KUKA KRL program: EPS_2_25252_PD2_A_20250910061714.src

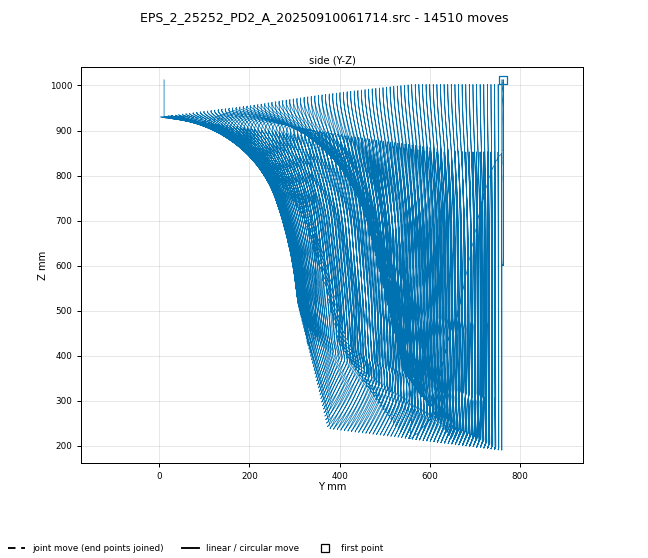
[picture p0: tool path of EPS_2_25252_PD2_A_20250910061714.src, 14510 of 14512 moves have a stored position in this frame; points joined in program order, loops and branches not executed]
&ACCESS RVP
&REL 4
&COMMENT QRS 19112012
&PARAM EDITMASK = *
DEF PART()
EXT BAS (BAS_COMMAND :IN,REAL :IN )
INT I
BAS (#INITMOV,0 )

;KUKA QRS Post kuka4.cps  Date:22-06-2017 !

File_ID=2827

QRS_PRE_INIT()

;Init var - Until changes are made in qrs_pre_init
Outlet_Square_prg=0
Inlet_1_Square_prg=0
Inlet_2_Square_prg=0
Inlet_3_Square_prg=0
Inlet_4_Square_prg=0
Inlet_5_Square_prg=0

Outlet_1={X 0.000, Y 562.000, Z 659.500, B 0.000, E1 0.000 }
Inlet_1={X 0.000, Y 675.710, Z 469.500, B 0.000, E1 90.000 }
Inlet_2={X 0.000, Y 612.000, Z 586.000, B 0.000, E1 180.000 }
Outlet_1_type=686
Inlet_1_type=366
Inlet_2_type=533
;QRS#1=Sidecore dimensions
;QRS#2=675-27" Concrete
;QRS#3=375-15" PVC SDR 35
;QRS#4=525-21" Concrete
;QRS#5=
;QRS#6=
;QRS#7=
;QRS#8=
;QRS#9=S306-38L
;QRS#10=20Y PSX
;QRS#11=S306-32
;QRS#12=
;QRS#13=
;QRS#14=
;QRS#15=
;QRS#16=1524x152x1448 4,75'
;QRS#17=EPS Height
;QRS#18=1002,5
;QRS#19=*
;QRS#20= UPDATED VERSION 22-06-2017
;QRS#21=*
Outlet_Square=0550
Inlet_1_Square=0250
Inlet_2_Square=0350
Inlet_3_Square=0
Inlet_4_Square=0
Inlet_5_Square=0
Mill_Square=1
Outlet_Square_Prg=265
Inlet_1_Square_prg=252
Inlet_2_Square_prg=263

QRS_INIT()

$ADVANCE=5

; T1
PTP {E1 177.625,E2 177.625}
PTP {X 0,Y 762.863,A -85,B 0,C 180,E1 177.625,E2 177.625,E3 0,E4 0,E5 0,E6 0}
QRS_SPEED_INIT()
LIN {X 0,Y 762.863,Z 1012.5,A -85,B 0,C 180,E1 177.625,E2 177.625,E3 0,E4 0,E5 0,E6 0} C_VEL
LIN {X 0,Y 762.863,Z 865.307,A -85,B 0,C 180,E1 177.625,E2 177.625} C_VEL
LIN {X 0,Y 762.863,Z 857.515,A -85,B 0,C 180,E1 177.625,E2 177.625} C_VEL
LIN {X 0,Y 762.89,Z 855.523,A -85,B 0,C 180,E1 177.789,E2 177.789} C_VEL
LIN {X 0,Y 763.311,Z 857.103,A -85,B 0,C 180,E1 179.062,E2 179.062} C_VEL
LIN {X 0,Y 763.552,Z 857.314,A -85,B 0,C 180,E1 179.437,E2 179.437} C_VEL
LIN {X 0,Y 763.78,Z 857.385,A -85,B 0,C 180,E1 180.187,E2 180.187} C_VEL
LIN {X 0,Y 763.382,Z 857.021,A -85,B 0,C 180,E1 180.938,E2 180.938} C_VEL
LIN {X 0,Y 763.064,Z 855.901,A -85,B 0,C 180,E1 181.878,E2 181.878} C_VEL
LIN {X 0,Y 763.224,Z 854.049,A -85,B 0,C 180,E1 182.816,E2 182.816} C_VEL
LIN {X 0,Y 763.674,Z 851.777,A -85,B 0,C 180,E1 183.621,E2 183.621} C_VEL
LIN {X 0,Y 763.795,Z 849.977,A -85,B 0,C 180,E1 184.156,E2 184.156} C_VEL
LIN {X 0,Y 763.342,Z 846.94,A -85,B 0,C 180,E1 184.931,E2 184.931} C_VEL
LIN {X 0,Y 763.012,Z 843.639,A -85,B 0,C 180,E1 185.64,E2 185.64} C_VEL
LIN {X 0,Y 763,Z 839.822,A -85,B 0,C 180,E1 186.347,E2 186.347} C_VEL
LIN {X 0,Y 763.321,Z 835.459,A -85,B 0,C 180,E1 187.053,E2 187.053} C_VEL
LIN {X 0,Y 763.757,Z 830.521,A -85,B 0,C 180,E1 187.758,E2 187.758} C_VEL
LIN {X 0,Y 763.804,Z 826.923,A -85,B 0,C 180,E1 188.231,E2 188.231} C_VEL
LIN {X 0,Y 763.447,Z 819.835,A -85,B 0,C 180,E1 189.065,E2 189.065} C_VEL
LIN {X 0,Y 763.299,Z 814.185,A -85,B 0,C 180,E1 189.661,E2 189.661} C_VEL
LIN {X 0,Y 763.415,Z 807.963,A -85,B 0,C 180,E1 190.255,E2 190.255} C_VEL
LIN {X 0,Y 763.624,Z 802.554,A -85,B 0,C 180,E1 190.729,E2 190.729} C_VEL
LIN {X 0,Y 763.851,Z 795.117,A -85,B 0,C 180,E1 191.322,E2 191.322} C_VEL
LIN {X 0,Y 763.76,Z 788.602,A -85,B 0,C 180,E1 191.802,E2 191.802} C_VEL
LIN {X 0,Y 763.573,Z 781.49,A -85,B 0,C 180,E1 192.284,E2 192.284} C_VEL
LIN {X 0,Y 763.481,Z 774.931,A -85,B 0,C 180,E1 192.694,E2 192.694} C_VEL
LIN {X 0,Y 763.571,Z 767.346,A -85,B 0,C 180,E1 193.125,E2 193.125} C_VEL
LIN {X 0,Y 763.752,Z 758.954,A -85,B 0,C 180,E1 193.555,E2 193.555} C_VEL
LIN {X 0,Y 763.785,Z 751.25,A -85,B 0,C 180,E1 193.917,E2 193.917} C_VEL
LIN {X 0,Y 763.828,Z 741.459,A -85,B 0,C 180,E1 194.328,E2 194.328} C_VEL
LIN {X 0,Y 763.759,Z 733.415,A -85,B 0,C 180,E1 194.632,E2 194.632} C_VEL
LIN {X 0,Y 763.747,Z 724.359,A -85,B 0,C 180,E1 194.936,E2 194.936} C_VEL
LIN {X 0,Y 763.826,Z 715.053,A -85,B 0,C 180,E1 195.207,E2 195.207} C_VEL
LIN {X 0,Y 763.801,Z 705.091,A -85,B 0,C 180,E1 195.458,E2 195.458} C_VEL
LIN {X 0,Y 763.852,Z 696.194,A -85,B 0,C 180,E1 195.647,E2 195.647} C_VEL
LIN {X 0,Y 763.86,Z 686.714,A -85,B 0,C 180,E1 195.814,E2 195.814} C_VEL
LIN {X 0,Y 763.829,Z 678.167,A -85,B 0,C 180,E1 195.936,E2 195.936} C_VEL
LIN {X 0,Y 763.809,Z 660.489,A -85,B 0,C 180,E1 196.119,E2 196.119} C_VEL
LIN {X 0,Y 763.591,Z 638.669,A -85,B 0,C 180,E1 196.333,E2 196.333} C_VEL
LIN {X 0,Y 763.668,Z 601.31,A -85,B 0,C 180,E1 197.602,E2 197.602} C_VEL
LIN {X 0,Y 763.856,Z 601.31,A -85,B 0,C 180,E1 200.095,E2 200.095} C_VEL
LIN {X 0,Y 763.798,Z 601.31,A -85,B 0,C 180,E1 208.326,E2 208.326} C_VEL
LIN {X 0,Y 762.387,Z 601.31,A -85,B 0,C 180,E1 210.541,E2 210.541} C_VEL
LIN {X 0,Y 762.703,Z 601.31,A -85,B 0,C 180,E1 214.993,E2 214.993} C_VEL
LIN {X 0,Y 763.707,Z 601.31,A -85,B 0,C 180,E1 216.696,E2 216.696} C_VEL
LIN {X 0,Y 763.72,Z 601.31,A -85,B 0,C 180,E1 224.719,E2 224.719} C_VEL
LIN {X 0,Y 763.504,Z 601.31,A -85,B 0,C 180,E1 225.265,E2 225.265} C_VEL
LIN {X 0,Y 762.431,Z 601.31,A -85,B 0,C 180,E1 230.388,E2 230.388} C_VEL
LIN {X 0,Y 763.803,Z 601.31,A -85,B 0,C 180,E1 232.744,E2 232.744} C_VEL
LIN {X 0,Y 763.78,Z 601.31,A -85,B 0,C 180,E1 239.845,E2 239.845} C_VEL
LIN {X 0,Y 763.759,Z 601.31,A -85,B 0,C 180,E1 240.061,E2 240.061} C_VEL
LIN {X 0,Y 763.232,Z 601.31,A -85,B 0,C 180,E1 240.149,E2 240.149} C_VEL
LIN {X 0,Y 763.551,Z 649.404,A -85,B 0,C 180,E1 240.674,E2 240.674} C_VEL
LIN {X 0,Y 763.815,Z 684.428,A -85,B 0,C 180,E1 241.063,E2 241.063} C_VEL
LIN {X 0,Y 763.833,Z 699.23,A -85,B 0,C 180,E1 241.258,E2 241.258} C_VEL
LIN {X 0,Y 763.72,Z 715.993,A -85,B 0,C 180,E1 241.54,E2 241.54} C_VEL
LIN {X 0,Y 763.487,Z 727.212,A -85,B 0,C 180,E1 241.761,E2 241.761} C_VEL
LIN {X 0,Y 763.725,Z 739.829,A -85,B 0,C 180,E1 242.069,E2 242.069} C_VEL
LIN {X 0,Y 763.771,Z 748.863,A -85,B 0,C 180,E1 242.303,E2 242.303} C_VEL
LIN {X 0,Y 763.77,Z 763.638,A -85,B 0,C 180,E1 242.732,E2 242.732} C_VEL
LIN {X 0,Y 763.697,Z 781.216,A -85,B 0,C 180,E1 243.321,E2 243.321} C_VEL
LIN {X 0,Y 763.6,Z 789.955,A -85,B 0,C 180,E1 243.645,E2 243.645} C_VEL
LIN {X 0,Y 763.691,Z 798.571,A -85,B 0,C 180,E1 243.99,E2 243.99} C_VEL
LIN {X 0,Y 763.619,Z 811.78,A -85,B 0,C 180,E1 244.551,E2 244.551} C_VEL
LIN {X 0,Y 763.589,Z 826.422,A -85,B 0,C 180,E1 245.241,E2 245.241} C_VEL
LIN {X 0,Y 763.713,Z 840.578,A -85,B 0,C 180,E1 245.981,E2 245.981} C_VEL
LIN {X 0,Y 763.688,Z 854.073,A -85,B 0,C 180,E1 246.747,E2 246.747} C_VEL
LIN {X 0,Y 763.544,Z 866.427,A -85,B 0,C 180,E1 247.506,E2 247.506} C_VEL
LIN {X 0,Y 763.324,Z 879.551,A -85,B 0,C 180,E1 248.385,E2 248.385} C_VEL
LIN {X 0,Y 763.405,Z 891.553,A -85,B 0,C 180,E1 249.267,E2 249.267} C_VEL
LIN {X 0,Y 763.694,Z 903.235,A -85,B 0,C 180,E1 250.204,E2 250.204} C_VEL
LIN {X 0,Y 763.727,Z 910.839,A -85,B 0,C 180,E1 250.857,E2 250.857} C_VEL
LIN {X 0,Y 763.444,Z 918.944,A -85,B 0,C 180,E1 251.586,E2 251.586} C_VEL
LIN {X 0,Y 763.19,Z 925.901,A -85,B 0,C 180,E1 252.243,E2 252.243} C_VEL
LIN {X 0,Y 763.133,Z 935.473,A -85,B 0,C 180,E1 253.224,E2 253.224} C_VEL
LIN {X 0,Y 763.43,Z 944.365,A -85,B 0,C 180,E1 254.22,E2 254.22} C_VEL
LIN {X 0,Y 763.797,Z 951.479,A -85,B 0,C 180,E1 255.09,E2 255.09} C_VEL
LIN {X 0,Y 763.66,Z 955.119,A -85,B 0,C 180,E1 255.556,E2 255.556} C_VEL
LIN {X 0,Y 763.118,Z 962.759,A -85,B 0,C 180,E1 256.586,E2 256.586} C_VEL
LIN {X 0,Y 762.806,Z 970.221,A -85,B 0,C 180,E1 257.703,E2 257.703} C_VEL
LIN {X 0,Y 763.093,Z 977.341,A -85,B 0,C 180,E1 258.905,E2 258.905} C_VEL
LIN {X 0,Y 763.744,Z 983.625,A -85,B 0,C 180,E1 260.107,E2 260.107} C_VEL
LIN {X 0,Y 763.847,Z 984.734,A -85,B 0,C 180,E1 260.346,E2 260.346} C_VEL
LIN {X 0,Y 763.274,Z 989.117,A -85,B 0,C 180,E1 261.289,E2 261.289} C_VEL
LIN {X 0,Y 762.776,Z 993.85,A -85,B 0,C 180,E1 262.468,E2 262.468} C_VEL
LIN {X 0,Y 762.955,Z 998.504,A -85,B 0,C 180,E1 263.888,E2 263.888} C_VEL
LIN {X 0,Y 763.445,Z 1001.065,A -85,B 0,C 180,E1 264.834,E2 264.834} C_VEL
LIN {X 0,Y 763.752,Z 1002.127,A -85,B 0,C 180,E1 265.307,E2 265.307} C_VEL
LIN {X 0,Y 763.413,Z 1004.112,A -85,B 0,C 180,E1 266.245,E2 266.245} C_VEL
LIN {X 0,Y 762.878,Z 1005.536,A -85,B 0,C 180,E1 267.183,E2 267.183} C_VEL
LIN {X 0,Y 762.652,Z 1006.74,A -85,B 0,C 180,E1 268.315,E2 268.315} C_VEL
LIN {X 0,Y 762.792,Z 1007.219,A -85,B 0,C 180,E1 269.061,E2 269.061} C_VEL
LIN {X 0,Y 763.864,Z 1007.171,A -85,B 0,C 180,E1 270.937,E2 270.937} C_VEL
LIN {X 0,Y 763.506,Z 1006.761,A -85,B 0,C 180,E1 271.626,E2 271.626} C_VEL
LIN {X 0,Y 763.098,Z 1005.877,A -85,B 0,C 180,E1 272.585,E2 272.585} C_VEL
LIN {X 0,Y 763.034,Z 1004.125,A -85,B 0,C 180,E1 273.756,E2 273.756} C_VEL
LIN {X 0,Y 763.619,Z 1001.06,A -85,B 0,C 180,E1 275.164,E2 275.164} C_VEL
LIN {X 0,Y 763.871,Z 999.763,A -85,B 0,C 180,E1 275.633,E2 275.633} C_VEL
LIN {X 0,Y 763.32,Z 997.027,A -85,B 0,C 180,E1 276.581,E2 276.581} C_VEL
LIN {X 0,Y 762.845,Z 993.851,A -85,B 0,C 180,E1 277.531,E2 277.531} C_VEL
LIN {X 0,Y 762.834,Z 988.065,A -85,B 0,C 180,E1 278.953,E2 278.953} C_VEL
LIN {X 0,Y 763.409,Z 982.441,A -85,B 0,C 180,E1 280.135,E2 280.135} C_VEL
LIN {X 0,Y 763.842,Z 978.617,A -85,B 0,C 180,E1 280.845,E2 280.845} C_VEL
LIN {X 0,Y 763.475,Z 974.56,A -85,B 0,C 180,E1 281.567,E2 281.567} C_VEL
LIN {X 0,Y 762.978,Z 968.584,A -85,B 0,C 180,E1 282.553,E2 282.553} C_VEL
LIN {X 0,Y 762.85,Z 960.441,A -85,B 0,C 180,E1 283.748,E2 283.748} C_VEL
LIN {X 0,Y 763.269,Z 952.013,A -85,B 0,C 180,E1 284.856,E2 284.856} C_VEL
LIN {X 0,Y 763.798,Z 943.48,A -85,B 0,C 180,E1 285.876,E2 285.876} C_VEL
LIN {X 0,Y 763.424,Z 933.185,A -85,B 0,C 180,E1 287.014,E2 287.014} C_VEL
LIN {X 0,Y 763.153,Z 923.436,A -85,B 0,C 180,E1 288.004,E2 288.004} C_VEL
LIN {X 0,Y 763.309,Z 911.702,A -85,B 0,C 180,E1 289.081,E2 289.081} C_VEL
LIN {X 0,Y 763.648,Z 901.038,A -85,B 0,C 180,E1 289.977,E2 289.977} C_VEL
LIN {X 0,Y 763.74,Z 891.15,A -85,B 0,C 180,E1 290.756,E2 290.756} C_VEL
LIN {X 0,Y 763.498,Z 877.794,A -85,B 0,C 180,E1 291.733,E2 291.733} C_VEL
LIN {X 0,Y 763.446,Z 864.411,A -85,B 0,C 180,E1 292.624,E2 292.624} C_VEL
LIN {X 0,Y 763.624,Z 850.805,A -85,B 0,C 180,E1 293.446,E2 293.446} C_VEL
LIN {X 0,Y 763.68,Z 836.999,A -85,B 0,C 180,E1 294.213,E2 294.213} C_VEL
LIN {X 0,Y 763.702,Z 822.332,A -85,B 0,C 180,E1 294.955,E2 294.955} C_VEL
LIN {X 0,Y 763.621,Z 807.81,A -85,B 0,C 180,E1 295.625,E2 295.625} C_VEL
LIN {X 0,Y 763.676,Z 793.458,A -85,B 0,C 180,E1 296.221,E2 296.221} C_VEL
LIN {X 0,Y 763.623,Z 777.576,A -85,B 0,C 180,E1 296.812,E2 296.812} C_VEL
LIN {X 0,Y 763.541,Z 771.61,A -85,B 0,C 180,E1 297.013,E2 297.013} C_VEL
LIN {X 0,Y 763.734,Z 760.339,A -85,B 0,C 180,E1 297.368,E2 297.368} C_VEL
LIN {X 0,Y 763.776,Z 744.554,A -85,B 0,C 180,E1 297.812,E2 297.812} C_VEL
LIN {X 0,Y 763.736,Z 728.036,A -85,B 0,C 180,E1 298.212,E2 298.212} C_VEL
LIN {X 0,Y 763.451,Z 711.795,A -85,B 0,C 180,E1 298.55,E2 298.55} C_VEL
LIN {X 0,Y 763.682,Z 694.79,A -85,B 0,C 180,E1 298.813,E2 298.813} C_VEL
LIN {X 0,Y 763.667,Z 674.795,A -85,B 0,C 180,E1 299.053,E2 299.053} C_VEL
LIN {X 0,Y 763.245,Z 602.276,A -85,B 0,C 180,E1 299.838,E2 299.838} C_VEL
LIN {X 0,Y 763.307,Z 601.31,A -85,B 0,C 180,E1 299.858,E2 299.858} C_VEL
LIN {X 0,Y 763.723,Z 601.31,A -85,B 0,C 180,E1 299.929,E2 299.929} C_VEL
LIN {X 0,Y 763.822,Z 601.31,A -85,B 0,C 180,E1 300.149,E2 300.149} C_VEL
LIN {X 0,Y 763.79,Z 601.31,A -85,B 0,C 180,E1 304.936,E2 304.936} C_VEL
LIN {X 0,Y 762.495,Z 601.31,A -85,B 0,C 180,E1 309.732,E2 309.732} C_VEL
LIN {X 0,Y 763.786,Z 601.31,A -85,B 0,C 180,E1 312.132,E2 312.132} C_VEL
LIN {X 0,Y 763.614,Z 601.31,A -85,B 0,C 180,E1 312.57,E2 312.57} C_VEL
LIN {X 0,Y 763.854,Z 601.31,A -85,B 0,C 180,E1 320.259,E2 320.259} C_VEL
LIN {X 0,Y 763.733,Z 601.31,A -85,B 0,C 180,E1 326.566,E2 326.566} C_VEL
LIN {X 0,Y 763.485,Z 601.31,A -85,B 0,C 180,E1 327.305,E2 327.305} C_VEL
LIN {X 0,Y 763.791,Z 601.31,A -85,B 0,C 180,E1 333.783,E2 333.783} C_VEL
LIN {X 0,Y 763.817,Z 601.31,A -85,B 0,C 180,E1 341.889,E2 341.889} C_VEL
LIN {X 0,Y 763.825,Z 601.31,A -85,B 0,C 180,E1 349.632,E2 349.632} C_VEL
LIN {X 0,Y 763.858,Z 601.31,A -85,B 0,C 180,E1 357.187,E2 357.187} C_VEL
LIN {X 0,Y 763.862,Z 601.31,A -85,B 0,C 180,E1 364.692,E2 364.692} C_VEL
LIN {X 0,Y 763.839,Z 601.31,A -85,B 0,C 180,E1 372.28,E2 372.28} C_VEL
LIN {X 0,Y 763.83,Z 601.31,A -85,B 0,C 180,E1 380.095,E2 380.095} C_VEL
LIN {X 0,Y 763.817,Z 601.31,A -85,B 0,C 180,E1 388.325,E2 388.325} C_VEL
LIN {X 0,Y 762.039,Z 601.31,A -85,B 0,C 180,E1 393.241,E2 393.241} C_VEL
LIN {X 0,Y 762.697,Z 601.31,A -85,B 0,C 180,E1 394.994,E2 394.994} C_VEL
LIN {X 0,Y 763.698,Z 601.31,A -85,B 0,C 180,E1 396.695,E2 396.695} C_VEL
LIN {X 0,Y 763.727,Z 601.31,A -85,B 0,C 180,E1 404.718,E2 404.718} C_VEL
LIN {X 0,Y 763.509,Z 601.31,A -85,B 0,C 180,E1 405.266,E2 405.266} C_VEL
LIN {X 0,Y 762.413,Z 601.31,A -85,B 0,C 180,E1 410.39,E2 410.39} C_VEL
LIN {X 0,Y 763.781,Z 601.31,A -85,B 0,C 180,E1 412.743,E2 412.743} C_VEL
LIN {X 0,Y 763.812,Z 601.31,A -85,B 0,C 180,E1 419.522,E2 419.522} C_VEL
LIN {X 0,Y 763.566,Z 601.31,A -85,B 0,C 180,E1 426.715,E2 426.715} C_VEL
LIN {X 0,Y 763.593,Z 601.31,A -85,B 0,C 180,E1 427.187,E2 427.187} C_VEL
LIN {X 0,Y 762.639,Z 601.31,A -85,B 0,C 180,E1 427.3,E2 427.3} C_VEL
LIN {X 0,Y 763.453,Z 613.717,A -85,B 0,C 180,E1 427.49,E2 427.49} C_VEL
LIN {X 0,Y 763.724,Z 626.926,A -85,B 0,C 180,E1 427.717,E2 427.717} C_VEL
LIN {X 0,Y 763.789,Z 639.679,A -85,B 0,C 180,E1 427.979,E2 427.979} C_VEL
LIN {X 0,Y 763.776,Z 651.564,A -85,B 0,C 180,E1 428.263,E2 428.263} C_VEL
LIN {X 0,Y 763.642,Z 664.747,A -85,B 0,C 180,E1 428.628,E2 428.628} C_VEL
LIN {X 0,Y 763.763,Z 676.879,A -85,B 0,C 180,E1 429.02,E2 429.02} C_VEL
LIN {X 0,Y 763.692,Z 689.935,A -85,B 0,C 180,E1 429.494,E2 429.494} C_VEL
LIN {X 0,Y 763.704,Z 701.321,A -85,B 0,C 180,E1 429.958,E2 429.958} C_VEL
LIN {X 0,Y 763.78,Z 713.403,A -85,B 0,C 180,E1 430.507,E2 430.507} C_VEL
LIN {X 0,Y 763.744,Z 724.924,A -85,B 0,C 180,E1 431.083,E2 431.083} C_VEL
LIN {X 0,Y 763.624,Z 736.787,A -85,B 0,C 180,E1 431.738,E2 431.738} C_VEL
LIN {X 0,Y 763.515,Z 745.388,A -85,B 0,C 180,E1 432.251,E2 432.251} C_VEL
LIN {X 0,Y 763.577,Z 756.581,A -85,B 0,C 180,E1 432.989,E2 432.989} C_VEL
LIN {X 0,Y 763.781,Z 766.757,A -85,B 0,C 180,E1 433.728,E2 433.728} C_VEL
LIN {X 0,Y 763.734,Z 775.073,A -85,B 0,C 180,E1 434.376,E2 434.376} C_VEL
LIN {X 0,Y 763.38,Z 783.89,A -85,B 0,C 180,E1 435.117,E2 435.117} C_VEL
LIN {X 0,Y 763.135,Z 792.692,A -85,B 0,C 180,E1 435.929,E2 435.929} C_VEL
LIN {X 0,Y 763.213,Z 800.042,A -85,B 0,C 180,E1 436.669,E2 436.669} C_VEL
LIN {X 0,Y 763.601,Z 808.027,A -85,B 0,C 180,E1 437.558,E2 437.558} C_VEL
LIN {X 0,Y 763.841,Z 813.343,A -85,B 0,C 180,E1 438.199,E2 438.199} C_VEL
LIN {X 0,Y 763.358,Z 820.655,A -85,B 0,C 180,E1 439.148,E2 439.148} C_VEL
LIN {X 0,Y 762.982,Z 827.171,A -85,B 0,C 180,E1 440.097,E2 440.097} C_VEL
LIN {X 0,Y 763.039,Z 832.95,A -85,B 0,C 180,E1 441.049,E2 441.049} C_VEL
LIN {X 0,Y 763.49,Z 838.043,A -85,B 0,C 180,E1 442.003,E2 442.003} C_VEL
LIN {X 0,Y 763.847,Z 841.371,A -85,B 0,C 180,E1 442.716,E2 442.716} C_VEL
LIN {X 0,Y 763.45,Z 844.408,A -85,B 0,C 180,E1 443.42,E2 443.42} C_VEL
LIN {X 0,Y 763.18,Z 846.302,A -85,B 0,C 180,E1 443.89,E2 443.89} C_VEL
LIN {X 0,Y 762.856,Z 849.53,A -85,B 0,C 180,E1 444.831,E2 444.831} C_VEL
LIN {X 0,Y 763.052,Z 852.685,A -85,B 0,C 180,E1 445.96,E2 445.96} C_VEL
LIN {X 0,Y 763.753,Z 855.112,A -85,B 0,C 180,E1 447.186,E2 447.186} C_VEL
LIN {X 0,Y 763.548,Z 856.237,A -85,B 0,C 180,E1 447.937,E2 447.937} C_VEL
LIN {X 0,Y 762.891,Z 857.232,A -85,B 0,C 180,E1 449.062,E2 449.062} C_VEL
LIN {X 0,Y 762.996,Z 857.194,A -85,B 0,C 180,E1 450.939,E2 450.939} C_VEL
LIN {X 0,Y 763.457,Z 856.519,A -85,B 0,C 180,E1 451.689,E2 451.689} C_VEL
LIN {X 0,Y 763.608,Z 854.985,A -85,B 0,C 180,E1 452.814,E2 452.814} C_VEL
LIN {X 0,Y 762.972,Z 852.552,A -85,B 0,C 180,E1 454.001,E2 454.001} C_VEL
LIN {X 0,Y 762.867,Z 850.661,A -85,B 0,C 180,E1 454.698,E2 454.698} C_VEL
LIN {X 0,Y 763.096,Z 847.645,A -85,B 0,C 180,E1 455.639,E2 455.639} C_VEL
LIN {X 0,Y 763.607,Z 844.044,A -85,B 0,C 180,E1 456.578,E2 456.578} C_VEL
LIN {X 0,Y 763.863,Z 842.053,A -85,B 0,C 180,E1 457.048,E2 457.048} C_VEL
LIN {X 0,Y 763.388,Z 837.561,A -85,B 0,C 180,E1 457.999,E2 457.999} C_VEL
LIN {X 0,Y 763.01,Z 832.407,A -85,B 0,C 180,E1 458.952,E2 458.952} C_VEL
LIN {X 0,Y 763.055,Z 826.56,A -85,B 0,C 180,E1 459.902,E2 459.902} C_VEL
LIN {X 0,Y 763.496,Z 819.973,A -85,B 0,C 180,E1 460.85,E2 460.85} C_VEL
LIN {X 0,Y 763.851,Z 814.56,A -85,B 0,C 180,E1 461.561,E2 461.561} C_VEL
LIN {X 0,Y 763.411,Z 805.949,A -85,B 0,C 180,E1 462.592,E2 462.592} C_VEL
LIN {X 0,Y 763.116,Z 797.827,A -85,B 0,C 180,E1 463.469,E2 463.469} C_VEL
LIN {X 0,Y 763.167,Z 790.215,A -85,B 0,C 180,E1 464.219,E2 464.219} C_VEL
LIN {X 0,Y 763.551,Z 780.772,A -85,B 0,C 180,E1 465.06,E2 465.06} C_VEL
LIN {X 0,Y 763.786,Z 772.241,A -85,B 0,C 180,E1 465.759,E2 465.759} C_VEL
LIN {X 0,Y 763.672,Z 763.931,A -85,B 0,C 180,E1 466.397,E2 466.397} C_VEL
LIN {X 0,Y 763.452,Z 753.435,A -85,B 0,C 180,E1 467.136,E2 467.136} C_VEL
LIN {X 0,Y 763.432,Z 742.882,A -85,B 0,C 180,E1 467.813,E2 467.813} C_VEL
LIN {X 0,Y 763.629,Z 732.669,A -85,B 0,C 180,E1 468.408,E2 468.408} C_VEL
LIN {X 0,Y 763.748,Z 721.763,A -85,B 0,C 180,E1 468.99,E2 468.99} C_VEL
LIN {X 0,Y 763.776,Z 710.571,A -85,B 0,C 180,E1 469.537,E2 469.537} C_VEL
LIN {X 0,Y 763.679,Z 697.818,A -85,B 0,C 180,E1 470.1,E2 470.1} C_VEL
LIN {X 0,Y 763.694,Z 685.483,A -85,B 0,C 180,E1 470.584,E2 470.584} C_VEL
LIN {X 0,Y 763.756,Z 672.801,A -85,B 0,C 180,E1 471.024,E2 471.024} C_VEL
LIN {X 0,Y 763.656,Z 660.443,A -85,B 0,C 180,E1 471.407,E2 471.407} C_VEL
LIN {X 0,Y 763.818,Z 647.246,A -85,B 0,C 180,E1 471.753,E2 471.753} C_VEL
LIN {X 0,Y 763.833,Z 634.146,A -85,B 0,C 180,E1 472.049,E2 472.049} C_VEL
LIN {X 0,Y 763.831,Z 621.273,A -85,B 0,C 180,E1 472.29,E2 472.29} C_VEL
LIN {X 0,Y 763.727,Z 607.963,A -85,B 0,C 180,E1 472.492,E2 472.492} C_VEL
LIN {X 0,Y 763.443,Z 601.78,A -85,B 0,C 180,E1 472.574,E2 472.574} C_VEL
LIN {X 0,Y 763.321,Z 601.31,A -85,B 0,C 180,E1 472.594,E2 472.594} C_VEL
LIN {X 0,Y 763.424,Z 601.31,A -85,B 0,C 180,E1 472.759,E2 472.759} C_VEL
LIN {X 0,Y 762.937,Z 601.31,A -85,B 0,C 180,E1 476.249,E2 476.249} C_VEL
LIN {X 0,Y 763.845,Z 601.31,A -85,B 0,C 180,E1 478.324,E2 478.324} C_VEL
LIN {X 0,Y 762.047,Z 601.31,A -85,B 0,C 180,E1 483.242,E2 483.242} C_VEL
LIN {X 0,Y 762.711,Z 601.31,A -85,B 0,C 180,E1 484.993,E2 484.993} C_VEL
LIN {X 0,Y 763.72,Z 601.31,A -85,B 0,C 180,E1 486.697,E2 486.697} C_VEL
LIN {X 0,Y 763.748,Z 601.31,A -85,B 0,C 180,E1 494.717,E2 494.717} C_VEL
LIN {X 0,Y 763.532,Z 601.31,A -85,B 0,C 180,E1 495.267,E2 495.267} C_VEL
LIN {X 0,Y 762.433,Z 601.31,A -85,B 0,C 180,E1 500.388,E2 500.388} C_VEL
LIN {X 0,Y 763.807,Z 601.31,A -85,B 0,C 180,E1 502.744,E2 502.744} C_VEL
LIN {X 0,Y 763.794,Z 601.31,A -85,B 0,C 180,E1 509.521,E2 509.521} C_VEL
LIN {X 0,Y 763.794,Z 601.31,A -85,B 0,C 180,E1 515.855,E2 515.855} C_VEL
LIN {X 0,Y 763.311,Z 601.31,A -85,B 0,C 180,E1 522.34,E2 522.34} C_VEL
LIN {X 0,Y 763.596,Z 630.997,A -85,B 0,C 180,E1 523.503,E2 523.503} C_VEL
LIN {X 0,Y 763.782,Z 675.397,A -85,B 0,C 180,E1 523.941,E2 523.941} C_VEL
LIN {X 0,Y 763.733,Z 684.643,A -85,B 0,C 180,E1 524.063,E2 524.063} C_VEL
LIN {X 0,Y 763.831,Z 693.752,A -85,B 0,C 180,E1 524.217,E2 524.217} C_VEL
LIN {X 0,Y 763.791,Z 702.752,A -85,B 0,C 180,E1 524.399,E2 524.399} C_VEL
LIN {X 0,Y 763.731,Z 711.65,A -85,B 0,C 180,E1 524.611,E2 524.611} C_VEL
LIN {X 0,Y 763.755,Z 719.441,A -85,B 0,C 180,E1 524.825,E2 524.825} C_VEL
LIN {X 0,Y 763.831,Z 729.06,A -85,B 0,C 180,E1 525.129,E2 525.129} C_VEL
LIN {X 0,Y 763.796,Z 737.568,A -85,B 0,C 180,E1 525.43,E2 525.43} C_VEL
LIN {X 0,Y 763.775,Z 746.635,A -85,B 0,C 180,E1 525.793,E2 525.793} C_VEL
LIN {X 0,Y 763.751,Z 755.527,A -85,B 0,C 180,E1 526.19,E2 526.19} C_VEL
LIN {X 0,Y 763.567,Z 763.547,A -85,B 0,C 180,E1 526.584,E2 526.584} C_VEL
LIN {X 0,Y 763.449,Z 770.453,A -85,B 0,C 180,E1 526.955,E2 526.955} C_VEL
LIN {X 0,Y 763.526,Z 778.468,A -85,B 0,C 180,E1 527.432,E2 527.432} C_VEL
LIN {X 0,Y 763.752,Z 786.449,A -85,B 0,C 180,E1 527.958,E2 527.958} C_VEL
LIN {X 0,Y 763.854,Z 793.148,A -85,B 0,C 180,E1 528.439,E2 528.439} C_VEL
LIN {X 0,Y 763.691,Z 799.305,A -85,B 0,C 180,E1 528.914,E2 528.914} C_VEL
LIN {X 0,Y 763.419,Z 806.315,A -85,B 0,C 180,E1 529.507,E2 529.507} C_VEL
LIN {X 0,Y 763.312,Z 811.472,A -85,B 0,C 180,E1 529.982,E2 529.982} C_VEL
LIN {X 0,Y 763.402,Z 817.368,A -85,B 0,C 180,E1 530.578,E2 530.578} C_VEL
LIN {X 0,Y 763.605,Z 821.734,A -85,B 0,C 180,E1 531.056,E2 531.056} C_VEL
LIN {X 0,Y 763.881,Z 827.607,A -85,B 0,C 180,E1 531.77,E2 531.77} C_VEL
LIN {X 0,Y 763.496,Z 832.846,A -85,B 0,C 180,E1 532.476,E2 532.476} C_VEL
LIN {X 0,Y 763.198,Z 836.057,A -85,B 0,C 180,E1 532.946,E2 532.946} C_VEL
LIN {X 0,Y 762.985,Z 840.331,A -85,B 0,C 180,E1 533.652,E2 533.652} C_VEL
LIN {X 0,Y 763.11,Z 844.072,A -85,B 0,C 180,E1 534.361,E2 534.361} C_VEL
LIN {X 0,Y 763.363,Z 846.268,A -85,B 0,C 180,E1 534.834,E2 534.834} C_VEL
LIN {X 0,Y 763.807,Z 849.501,A -85,B 0,C 180,E1 535.624,E2 535.624} C_VEL
LIN {X 0,Y 763.791,Z 850.603,A -85,B 0,C 180,E1 535.941,E2 535.941} C_VEL
LIN {X 0,Y 763.396,Z 852.627,A -85,B 0,C 180,E1 536.571,E2 536.571} C_VEL
LIN {X 0,Y 763.05,Z 854.257,A -85,B 0,C 180,E1 537.184,E2 537.184} C_VEL
LIN {X 0,Y 762.89,Z 855.523,A -85,B 0,C 180,E1 537.789,E2 537.789} C_VEL
LIN {X 0,Y 762.867,Z 857.499,A -85,B 0,C 180,E1 537.916,E2 537.916} C_VEL
LIN {X 0,Y 762.867,Z 1012.5,A -85,B 0,C 180,E1 537.916,E2 537.916} C_VEL
LIN {X 0,Y 762.867,Z 1012.5,A -85,B 0,C 180,E1 537.916,E2 537.916}

QRS_NEXT_CUT()
PTP {E1 537.186,E2 537.186}
PTP {X 0,Y 759.911,A -85,B 0,C 180,E1 537.186,E2 537.186,E3 0,E4 0,E5 0,E6 0}
QRS_SPEED_INIT()
LIN {X 0,Y 759.911,Z 1012.5,A -85,B 0,C 180,E1 537.186,E2 537.186,E3 0,E4 0,E5 0,E6 0} C_VEL
LIN {X 0,Y 759.911,Z 859.359,A -85,B 0,C 180,E1 537.186,E2 537.186} C_VEL
LIN {X 0,Y 759.911,Z 850.88,A -85,B 0,C 180,E1 537.186,E2 537.186} C_VEL
LIN {X 0,Y 759.915,Z 848.921,A -85,B 0,C 180,E1 537.065,E2 537.065} C_VEL
LIN {X 0,Y 759.916,Z 844.691,A -85,B 0,C 180,E1 535.699,E2 535.699} C_VEL
LIN {X 0,Y 759.912,Z 838.727,A -85,B 0,C 180,E1 534.337,E2 534.337} C_VEL
LIN {X 0,Y 759.916,Z 830.826,A -85,B 0,C 180,E1 532.971,E2 532.971} C_VEL
LIN {X 0,Y 759.916,Z 821.375,A -85,B 0,C 180,E1 531.678,E2 531.678} C_VEL
LIN {X 0,Y 759.915,Z 810.407,A -85,B 0,C 180,E1 530.457,E2 530.457} C_VEL
LIN {X 0,Y 759.914,Z 797.91,A -85,B 0,C 180,E1 529.308,E2 529.308} C_VEL
LIN {X 0,Y 759.916,Z 783.678,A -85,B 0,C 180,E1 528.223,E2 528.223} C_VEL
LIN {X 0,Y 759.918,Z 768.565,A -85,B 0,C 180,E1 527.268,E2 527.268} C_VEL
LIN {X 0,Y 759.918,Z 753.017,A -85,B 0,C 180,E1 526.455,E2 526.455} C_VEL
LIN {X 0,Y 759.892,Z 736.694,A -85,B 0,C 180,E1 525.755,E2 525.755} C_VEL
LIN {X 0,Y 759.918,Z 719.642,A -85,B 0,C 180,E1 525.172,E2 525.172} C_VEL
LIN {X 0,Y 759.913,Z 702.22,A -85,B 0,C 180,E1 524.713,E2 524.713} C_VEL
LIN {X 0,Y 759.911,Z 683.596,A -85,B 0,C 180,E1 524.364,E2 524.364} C_VEL
LIN {X 0,Y 759.901,Z 658.001,A -85,B 0,C 180,E1 524.077,E2 524.077} C_VEL
LIN {X 0,Y 759.864,Z 469.775,A -85,B 0,C 180,E1 522.244,E2 522.244} C_VEL
LIN {X 0,Y 759.9,Z 416.635,A -85,B 0,C 180,E1 519.593,E2 519.593} C_VEL
LIN {X 0,Y 759.918,Z 361.495,A -85,B 0,C 180,E1 516.791,E2 516.791} C_VEL
LIN {X 0,Y 759.91,Z 307.45,A -85,B 0,C 180,E1 513.987,E2 513.987} C_VEL
LIN {X 0,Y 759.913,Z 254.157,A -85,B 0,C 180,E1 511.163,E2 511.163} C_VEL
LIN {X 0,Y 759.884,Z 202.297,A -85,B 0,C 180,E1 508.359,E2 508.359} C_VEL
LIN {X 0,Y 759.874,Z 190.577,A -85,B 0,C 180,E1 507.707,E2 507.707} C_VEL
LIN {X 0,Y 759.897,Z 190.571,A -85,B 0,C 180,E1 504.899,E2 504.899} C_VEL
LIN {X 0,Y 759.895,Z 190.577,A -85,B 0,C 180,E1 501.989,E2 501.989} C_VEL
LIN {X 0,Y 759.84,Z 190.578,A -85,B 0,C 180,E1 499.354,E2 499.354} C_VEL
LIN {X 0,Y 759.917,Z 190.569,A -85,B 0,C 180,E1 496.515,E2 496.515} C_VEL
LIN {X 0,Y 759.911,Z 190.578,A -85,B 0,C 180,E1 493.589,E2 493.589} C_VEL
LIN {X 0,Y 759.882,Z 190.572,A -85,B 0,C 180,E1 490.743,E2 490.743} C_VEL
LIN {X 0,Y 759.843,Z 190.578,A -85,B 0,C 180,E1 487.823,E2 487.823} C_VEL
LIN {X 0,Y 759.881,Z 190.577,A -85,B 0,C 180,E1 485.286,E2 485.286} C_VEL
LIN {X 0,Y 759.897,Z 190.758,A -85,B 0,C 180,E1 482.716,E2 482.716} C_VEL
LIN {X 0,Y 759.899,Z 231.312,A -85,B 0,C 180,E1 480.001,E2 480.001} C_VEL
LIN {X 0,Y 759.904,Z 273.516,A -85,B 0,C 180,E1 477.252,E2 477.252} C_VEL
LIN {X 0,Y 759.912,Z 304.464,A -85,B 0,C 180,E1 475.291,E2 475.291} C_VEL
LIN {X 0,Y 759.918,Z 592.91,A -85,B 0,C 180,E1 472.37,E2 472.37} C_VEL
LIN {X 0,Y 759.914,Z 615.626,A -85,B 0,C 180,E1 472.085,E2 472.085} C_VEL
LIN {X 0,Y 759.913,Z 637.423,A -85,B 0,C 180,E1 471.679,E2 471.679} C_VEL
LIN {X 0,Y 759.909,Z 657.419,A -85,B 0,C 180,E1 471.173,E2 471.173} C_VEL
LIN {X 0,Y 759.905,Z 678.887,A -85,B 0,C 180,E1 470.488,E2 470.488} C_VEL
LIN {X 0,Y 759.918,Z 698.468,A -85,B 0,C 180,E1 469.725,E2 469.725} C_VEL
LIN {X 0,Y 759.917,Z 717.218,A -85,B 0,C 180,E1 468.846,E2 468.846} C_VEL
LIN {X 0,Y 759.915,Z 736.006,A -85,B 0,C 180,E1 467.814,E2 467.814} C_VEL
LIN {X 0,Y 759.911,Z 753.642,A -85,B 0,C 180,E1 466.683,E2 466.683} C_VEL
LIN {X 0,Y 759.912,Z 770.137,A -85,B 0,C 180,E1 465.453,E2 465.453} C_VEL
LIN {X 0,Y 759.919,Z 785.295,A -85,B 0,C 180,E1 464.131,E2 464.131} C_VEL
LIN {X 0,Y 759.913,Z 798.741,A -85,B 0,C 180,E1 462.771,E2 462.771} C_VEL
LIN {X 0,Y 759.912,Z 811.161,A -85,B 0,C 180,E1 461.306,E2 461.306} C_VEL
LIN {X 0,Y 759.912,Z 821.569,A -85,B 0,C 180,E1 459.849,E2 459.849} C_VEL
LIN {X 0,Y 759.907,Z 830.684,A -85,B 0,C 180,E1 458.314,E2 458.314} C_VEL
LIN {X 0,Y 759.898,Z 838.372,A -85,B 0,C 180,E1 456.725,E2 456.725} C_VEL
LIN {X 0,Y 759.904,Z 844.26,A -85,B 0,C 180,E1 455.133,E2 455.133} C_VEL
LIN {X 0,Y 759.914,Z 848.686,A -85,B 0,C 180,E1 453.47,E2 453.47} C_VEL
LIN {X 0,Y 759.918,Z 851.442,A -85,B 0,C 180,E1 451.81,E2 451.81} C_VEL
LIN {X 0,Y 759.908,Z 852.45,A -85,B 0,C 180,E1 450.151,E2 450.151} C_VEL
LIN {X 0,Y 759.899,Z 851.787,A -85,B 0,C 180,E1 448.492,E2 448.492} C_VEL
LIN {X 0,Y 759.896,Z 849.505,A -85,B 0,C 180,E1 446.832,E2 446.832} C_VEL
LIN {X 0,Y 759.902,Z 845.701,A -85,B 0,C 180,E1 445.245,E2 445.245} C_VEL
LIN {X 0,Y 759.913,Z 840.243,A -85,B 0,C 180,E1 443.654,E2 443.654} C_VEL
LIN {X 0,Y 759.911,Z 833.15,A -85,B 0,C 180,E1 442.059,E2 442.059} C_VEL
LIN {X 0,Y 759.903,Z 824.561,A -85,B 0,C 180,E1 440.533,E2 440.533} C_VEL
LIN {X 0,Y 759.903,Z 814.081,A -85,B 0,C 180,E1 438.992,E2 438.992} C_VEL
LIN {X 0,Y 759.908,Z 802.385,A -85,B 0,C 180,E1 437.538,E2 437.538} C_VEL
LIN {X 0,Y 759.906,Z 789.125,A -85,B 0,C 180,E1 436.144,E2 436.144} C_VEL
LIN {X 0,Y 759.911,Z 774.48,A -85,B 0,C 180,E1 434.821,E2 434.821} C_VEL
LIN {X 0,Y 759.916,Z 757.861,A -85,B 0,C 180,E1 433.528,E2 433.528} C_VEL
LIN {X 0,Y 759.917,Z 740.817,A -85,B 0,C 180,E1 432.384,E2 432.384} C_VEL
LIN {X 0,Y 759.915,Z 722.406,A -85,B 0,C 180,E1 431.33,E2 431.33} C_VEL
LIN {X 0,Y 759.917,Z 703.45,A -85,B 0,C 180,E1 430.409,E2 430.409} C_VEL
LIN {X 0,Y 759.916,Z 683.635,A -85,B 0,C 180,E1 429.593,E2 429.593} C_VEL
LIN {X 0,Y 759.917,Z 662.813,A -85,B 0,C 180,E1 428.891,E2 428.891} C_VEL
LIN {X 0,Y 759.907,Z 642.122,A -85,B 0,C 180,E1 428.341,E2 428.341} C_VEL
LIN {X 0,Y 759.915,Z 621.37,A -85,B 0,C 180,E1 427.915,E2 427.915} C_VEL
LIN {X 0,Y 759.917,Z 600.246,A -85,B 0,C 180,E1 427.619,E2 427.619} C_VEL
LIN {X 0,Y 759.913,Z 307.626,A -85,B 0,C 180,E1 424.651,E2 424.651} C_VEL
LIN {X 0,Y 759.917,Z 303.957,A -85,B 0,C 180,E1 424.599,E2 424.599} C_VEL
LIN {X 0,Y 759.919,Z 257.758,A -85,B 0,C 180,E1 421.641,E2 421.641} C_VEL
LIN {X 0,Y 759.889,Z 216.102,A -85,B 0,C 180,E1 418.9,E2 418.9} C_VEL
LIN {X 0,Y 759.875,Z 190.573,A -85,B 0,C 180,E1 417.171,E2 417.171} C_VEL
LIN {X 0,Y 759.906,Z 190.578,A -85,B 0,C 180,E1 414.407,E2 414.407} C_VEL
LIN {X 0,Y 759.899,Z 190.566,A -85,B 0,C 180,E1 411.407,E2 411.407} C_VEL
LIN {X 0,Y 759.893,Z 190.575,A -85,B 0,C 180,E1 408.558,E2 408.558} C_VEL
LIN {X 0,Y 759.914,Z 190.565,A -85,B 0,C 180,E1 405.573,E2 405.573} C_VEL
LIN {X 0,Y 759.881,Z 190.572,A -85,B 0,C 180,E1 402.757,E2 402.757} C_VEL
LIN {X 0,Y 759.901,Z 190.573,A -85,B 0,C 180,E1 400.021,E2 400.021} C_VEL
LIN {X 0,Y 759.891,Z 190.567,A -85,B 0,C 180,E1 397.118,E2 397.118} C_VEL
LIN {X 0,Y 759.914,Z 190.578,A -85,B 0,C 180,E1 394.275,E2 394.275} C_VEL
LIN {X 0,Y 759.912,Z 190.564,A -85,B 0,C 180,E1 391.315,E2 391.315} C_VEL
LIN {X 0,Y 759.918,Z 190.577,A -85,B 0,C 180,E1 388.274,E2 388.274} C_VEL
LIN {X 0,Y 759.912,Z 190.564,A -85,B 0,C 180,E1 385.234,E2 385.234} C_VEL
LIN {X 0,Y 759.91,Z 190.577,A -85,B 0,C 180,E1 382.269,E2 382.269} C_VEL
LIN {X 0,Y 759.912,Z 190.564,A -85,B 0,C 180,E1 379.285,E2 379.285} C_VEL
LIN {X 0,Y 759.912,Z 190.577,A -85,B 0,C 180,E1 376.276,E2 376.276} C_VEL
LIN {X 0,Y 759.901,Z 190.565,A -85,B 0,C 180,E1 373.313,E2 373.313} C_VEL
LIN {X 0,Y 759.904,Z 190.574,A -85,B 0,C 180,E1 370.385,E2 370.385} C_VEL
LIN {X 0,Y 759.884,Z 190.57,A -85,B 0,C 180,E1 367.637,E2 367.637} C_VEL
LIN {X 0,Y 759.903,Z 190.566,A -85,B 0,C 180,E1 364.831,E2 364.831} C_VEL
LIN {X 0,Y 759.896,Z 190.575,A -85,B 0,C 180,E1 361.961,E2 361.961} C_VEL
LIN {X 0,Y 759.916,Z 190.563,A -85,B 0,C 180,E1 359.02,E2 359.02} C_VEL
LIN {X 0,Y 759.9,Z 190.576,A -85,B 0,C 180,E1 356.001,E2 356.001} C_VEL
LIN {X 0,Y 759.896,Z 190.565,A -85,B 0,C 180,E1 353.123,E2 353.123} C_VEL
LIN {X 0,Y 759.911,Z 190.578,A -85,B 0,C 180,E1 350.151,E2 350.151} C_VEL
LIN {X 0,Y 759.874,Z 190.57,A -85,B 0,C 180,E1 347.383,E2 347.383} C_VEL
LIN {X 0,Y 759.907,Z 190.569,A -85,B 0,C 180,E1 344.586,E2 344.586} C_VEL
LIN {X 0,Y 759.879,Z 190.574,A -85,B 0,C 180,E1 341.749,E2 341.749} C_VEL
LIN {X 0,Y 759.887,Z 190.567,A -85,B 0,C 180,E1 339.028,E2 339.028} C_VEL
LIN {X 0,Y 759.907,Z 190.577,A -85,B 0,C 180,E1 336.009,E2 336.009} C_VEL
LIN {X 0,Y 759.866,Z 190.57,A -85,B 0,C 180,E1 333.254,E2 333.254} C_VEL
LIN {X 0,Y 759.912,Z 190.568,A -85,B 0,C 180,E1 330.521,E2 330.521} C_VEL
LIN {X 0,Y 759.87,Z 190.574,A -85,B 0,C 180,E1 327.649,E2 327.649} C_VEL
LIN {X 0,Y 759.872,Z 190.569,A -85,B 0,C 180,E1 324.99,E2 324.99} C_VEL
LIN {X 0,Y 759.918,Z 190.577,A -85,B 0,C 180,E1 322.086,E2 322.086} C_VEL
LIN {X 0,Y 759.854,Z 190.573,A -85,B 0,C 180,E1 319.355,E2 319.355} C_VEL
LIN {X 0,Y 759.893,Z 190.568,A -85,B 0,C 180,E1 316.69,E2 316.69} C_VEL
LIN {X 0,Y 759.873,Z 190.576,A -85,B 0,C 180,E1 313.696,E2 313.696} C_VEL
LIN {X 0,Y 759.849,Z 190.572,A -85,B 0,C 180,E1 311.144,E2 311.144} C_VEL
LIN {X 0,Y 759.912,Z 190.569,A -85,B 0,C 180,E1 308.473,E2 308.473} C_VEL
LIN {X 0,Y 759.86,Z 190.667,A -85,B 0,C 180,E1 307.583,E2 307.583} C_VEL
LIN {X 0,Y 759.867,Z 242.061,A -85,B 0,C 180,E1 305.287,E2 305.287} C_VEL
LIN {X 0,Y 759.895,Z 298.787,A -85,B 0,C 180,E1 302.831,E2 302.831} C_VEL
LIN {X 0,Y 759.917,Z 557.126,A -85,B 0,C 180,E1 300.027,E2 300.027} C_VEL
LIN {X 0,Y 759.916,Z 689.995,A -85,B 0,C 180,E1 298.595,E2 298.595} C_VEL
LIN {X 0,Y 759.912,Z 714.301,A -85,B 0,C 180,E1 298.21,E2 298.21} C_VEL
LIN {X 0,Y 759.907,Z 735.677,A -85,B 0,C 180,E1 297.742,E2 297.742} C_VEL
LIN {X 0,Y 759.894,Z 755.109,A -85,B 0,C 180,E1 297.22,E2 297.22} C_VEL
LIN {X 0,Y 759.919,Z 777.739,A -85,B 0,C 180,E1 296.491,E2 296.491} C_VEL
LIN {X 0,Y 759.916,Z 799.252,A -85,B 0,C 180,E1 295.651,E2 295.651} C_VEL
LIN {X 0,Y 759.913,Z 818.66,A -85,B 0,C 180,E1 294.783,E2 294.783} C_VEL
LIN {X 0,Y 759.91,Z 841.061,A -85,B 0,C 180,E1 293.62,E2 293.62} C_VEL
LIN {X 0,Y 759.911,Z 859.706,A -85,B 0,C 180,E1 292.513,E2 292.513} C_VEL
LIN {X 0,Y 759.906,Z 879.524,A -85,B 0,C 180,E1 291.173,E2 291.173} C_VEL
LIN {X 0,Y 759.916,Z 896.886,A -85,B 0,C 180,E1 289.845,E2 289.845} C_VEL
LIN {X 0,Y 759.907,Z 913.391,A -85,B 0,C 180,E1 288.409,E2 288.409} C_VEL
LIN {X 0,Y 759.895,Z 927.948,A -85,B 0,C 180,E1 286.984,E2 286.984} C_VEL
LIN {X 0,Y 759.899,Z 942.876,A -85,B 0,C 180,E1 285.312,E2 285.312} C_VEL
LIN {X 0,Y 759.91,Z 954.559,A -85,B 0,C 180,E1 283.816,E2 283.816} C_VEL
LIN {X 0,Y 759.911,Z 966.786,A -85,B 0,C 180,E1 281.999,E2 281.999} C_VEL
LIN {X 0,Y 759.907,Z 975.555,A -85,B 0,C 180,E1 280.462,E2 280.462} C_VEL
LIN {X 0,Y 759.883,Z 984.074,A -85,B 0,C 180,E1 278.704,E2 278.704} C_VEL
LIN {X 0,Y 759.918,Z 990.726,A -85,B 0,C 180,E1 276.953,E2 276.953} C_VEL
LIN {X 0,Y 759.883,Z 995.51,A -85,B 0,C 180,E1 275.361,E2 275.361} C_VEL
LIN {X 0,Y 759.919,Z 999.559,A -85,B 0,C 180,E1 273.47,E2 273.47} C_VEL
LIN {X 0,Y 759.903,Z 1001.63,A -85,B 0,C 180,E1 271.81,E2 271.81} C_VEL
LIN {X 0,Y 759.92,Z 1002.5,A -85,B 0,C 180,E1 270,E2 270} C_VEL
LIN {X 0,Y 759.904,Z 1001.63,A -85,B 0,C 180,E1 268.19,E2 268.19} C_VEL
LIN {X 0,Y 759.919,Z 999.559,A -85,B 0,C 180,E1 266.53,E2 266.53} C_VEL
LIN {X 0,Y 759.883,Z 995.51,A -85,B 0,C 180,E1 264.639,E2 264.639} C_VEL
LIN {X 0,Y 759.918,Z 990.725,A -85,B 0,C 180,E1 263.047,E2 263.047} C_VEL
LIN {X 0,Y 759.884,Z 983.729,A -85,B 0,C 180,E1 261.22,E2 261.22} C_VEL
LIN {X 0,Y 759.907,Z 975.555,A -85,B 0,C 180,E1 259.538,E2 259.538} C_VEL
LIN {X 0,Y 759.911,Z 966.785,A -85,B 0,C 180,E1 258.001,E2 258.001} C_VEL
LIN {X 0,Y 759.909,Z 954.265,A -85,B 0,C 180,E1 256.144,E2 256.144} C_VEL
LIN {X 0,Y 759.9,Z 942.679,A -85,B 0,C 180,E1 254.664,E2 254.664} C_VEL
LIN {X 0,Y 759.896,Z 927.17,A -85,B 0,C 180,E1 252.937,E2 252.937} C_VEL
LIN {X 0,Y 759.903,Z 912.54,A -85,B 0,C 180,E1 251.512,E2 251.512} C_VEL
LIN {X 0,Y 759.917,Z 894.472,A -85,B 0,C 180,E1 249.964,E2 249.964} C_VEL
LIN {X 0,Y 759.91,Z 877.578,A -85,B 0,C 180,E1 248.684,E2 248.684} C_VEL
LIN {X 0,Y 759.913,Z 857.72,A -85,B 0,C 180,E1 247.364,E2 247.364} C_VEL
LIN {X 0,Y 759.91,Z 838.877,A -85,B 0,C 180,E1 246.257,E2 246.257} C_VEL
LIN {X 0,Y 759.913,Z 817.007,A -85,B 0,C 180,E1 245.14,E2 245.14} C_VEL
LIN {X 0,Y 759.917,Z 798.063,A -85,B 0,C 180,E1 244.299,E2 244.299} C_VEL
LIN {X 0,Y 759.912,Z 775.318,A -85,B 0,C 180,E1 243.425,E2 243.425} C_VEL
LIN {X 0,Y 759.895,Z 754.005,A -85,B 0,C 180,E1 242.748,E2 242.748} C_VEL
LIN {X 0,Y 759.906,Z 734.048,A -85,B 0,C 180,E1 242.218,E2 242.218} C_VEL
LIN {X 0,Y 759.917,Z 709.304,A -85,B 0,C 180,E1 241.7,E2 241.7} C_VEL
LIN {X 0,Y 759.916,Z 688.273,A -85,B 0,C 180,E1 241.383,E2 241.383} C_VEL
LIN {X 0,Y 759.868,Z 431.867,A -85,B 0,C 180,E1 238.623,E2 238.623} C_VEL
LIN {X 0,Y 759.895,Z 298.203,A -85,B 0,C 180,E1 237.151,E2 237.151} C_VEL
LIN {X 0,Y 759.867,Z 239.96,A -85,B 0,C 180,E1 234.621,E2 234.621} C_VEL
LIN {X 0,Y 759.906,Z 190.577,A -85,B 0,C 180,E1 232.405,E2 232.405} C_VEL
LIN {X 0,Y 759.909,Z 190.576,A -85,B 0,C 180,E1 229.512,E2 229.512} C_VEL
LIN {X 0,Y 759.908,Z 190.578,A -85,B 0,C 180,E1 226.689,E2 226.689} C_VEL
LIN {X 0,Y 759.915,Z 190.577,A -85,B 0,C 180,E1 223.797,E2 223.797} C_VEL
LIN {X 0,Y 759.909,Z 190.578,A -85,B 0,C 180,E1 220.94,E2 220.94} C_VEL
LIN {X 0,Y 759.907,Z 190.579,A -85,B 0,C 180,E1 218.106,E2 218.106} C_VEL
LIN {X 0,Y 759.919,Z 190.577,A -85,B 0,C 180,E1 215.192,E2 215.192} C_VEL
LIN {X 0,Y 759.911,Z 190.578,A -85,B 0,C 180,E1 212.291,E2 212.291} C_VEL
LIN {X 0,Y 759.904,Z 190.635,A -85,B 0,C 180,E1 212.113,E2 212.113} C_VEL
LIN {X 0,Y 759.914,Z 241.509,A -85,B 0,C 180,E1 209.393,E2 209.393} C_VEL
LIN {X 0,Y 759.875,Z 296.655,A -85,B 0,C 180,E1 206.492,E2 206.492} C_VEL
LIN {X 0,Y 759.873,Z 345.368,A -85,B 0,C 180,E1 203.95,E2 203.95} C_VEL
LIN {X 0,Y 759.905,Z 400.989,A -85,B 0,C 180,E1 201.107,E2 201.107} C_VEL
LIN {X 0,Y 759.874,Z 457.176,A -85,B 0,C 180,E1 198.29,E2 198.29} C_VEL
LIN {X 0,Y 759.867,Z 470.197,A -85,B 0,C 180,E1 197.65,E2 197.65} C_VEL
LIN {X 0,Y 759.915,Z 679.188,A -85,B 0,C 180,E1 195.612,E2 195.612} C_VEL
LIN {X 0,Y 759.914,Z 698.227,A -85,B 0,C 180,E1 195.287,E2 195.287} C_VEL
LIN {X 0,Y 759.916,Z 716.693,A -85,B 0,C 180,E1 194.828,E2 194.828} C_VEL
LIN {X 0,Y 759.892,Z 734.388,A -85,B 0,C 180,E1 194.245,E2 194.245} C_VEL
LIN {X 0,Y 759.918,Z 751.15,A -85,B 0,C 180,E1 193.545,E2 193.545} C_VEL
LIN {X 0,Y 759.917,Z 767.025,A -85,B 0,C 180,E1 192.732,E2 192.732} C_VEL
LIN {X 0,Y 759.916,Z 782.388,A -85,B 0,C 180,E1 191.777,E2 191.777} C_VEL
LIN {X 0,Y 759.918,Z 795.899,A -85,B 0,C 180,E1 190.769,E2 190.769} C_VEL
LIN {X 0,Y 759.918,Z 808.722,A -85,B 0,C 180,E1 189.62,E2 189.62} C_VEL
LIN {X 0,Y 759.913,Z 819.984,A -85,B 0,C 180,E1 188.398,E2 188.398} C_VEL
LIN {X 0,Y 759.919,Z 829.698,A -85,B 0,C 180,E1 187.105,E2 187.105} C_VEL
LIN {X 0,Y 759.911,Z 837.436,A -85,B 0,C 180,E1 185.815,E2 185.815} C_VEL
LIN {X 0,Y 759.91,Z 843.729,A -85,B 0,C 180,E1 184.453,E2 184.453} C_VEL
LIN {X 0,Y 759.916,Z 848.455,A -85,B 0,C 180,E1 183.017,E2 183.017} C_VEL
LIN {X 0,Y 759.909,Z 851.332,A -85,B 0,C 180,E1 181.583,E2 181.583} C_VEL
LIN {X 0,Y 759.911,Z 852.449,A -85,B 0,C 180,E1 180.151,E2 180.151} C_VEL
LIN {X 0,Y 759.915,Z 851.822,A -85,B 0,C 180,E1 178.718,E2 178.718} C_VEL
LIN {X 0,Y 759.911,Z 849.442,A -85,B 0,C 180,E1 177.285,E2 177.285} C_VEL
LIN {X 0,Y 759.915,Z 848.921,A -85,B 0,C 180,E1 177.065,E2 177.065} C_VEL
LIN {X 0,Y 758.934,Z 847.398,A -85,B 0,C 180,E1 176.498,E2 176.498} C_VEL
LIN {X 0,Y 753.637,Z 843.222,A -85,B 0,C 180,E1 175.285,E2 175.285} C_VEL
LIN {X 0,Y 752.012,Z 840.67,A -85,B 0,C 180,E1 174.69,E2 174.69} C_VEL
LIN {X 0,Y 751.92,Z 839.929,A -85,B 0,C 180,E1 174.529,E2 174.529} C_VEL
LIN {X 0,Y 751.924,Z 832.732,A -85,B 0,C 180,E1 173.203,E2 173.203} C_VEL
LIN {X 0,Y 751.931,Z 823.768,A -85,B 0,C 180,E1 171.897,E2 171.897} C_VEL
LIN {X 0,Y 751.951,Z 813.349,A -85,B 0,C 180,E1 170.664,E2 170.664} C_VEL
LIN {X 0,Y 751.972,Z 801.487,A -85,B 0,C 180,E1 169.504,E2 169.504} C_VEL
LIN {X 0,Y 752,Z 788.155,A -85,B 0,C 180,E1 168.418,E2 168.418} C_VEL
LIN {X 0,Y 752.038,Z 773.063,A -85,B 0,C 180,E1 167.398,E2 167.398} C_VEL
LIN {X 0,Y 752.076,Z 757.188,A -85,B 0,C 180,E1 166.515,E2 166.515} C_VEL
LIN {X 0,Y 752.089,Z 740.168,A -85,B 0,C 180,E1 165.742,E2 165.742} C_VEL
LIN {X 0,Y 752.14,Z 723.078,A -85,B 0,C 180,E1 165.121,E2 165.121} C_VEL
LIN {X 0,Y 752.176,Z 704.904,A -85,B 0,C 180,E1 164.614,E2 164.614} C_VEL
LIN {X 0,Y 752.196,Z 686.353,A -85,B 0,C 180,E1 164.242,E2 164.242} C_VEL
LIN {X 0,Y 752.21,Z 666.095,A -85,B 0,C 180,E1 163.989,E2 163.989} C_VEL
LIN {X 0,Y 752.136,Z 469.964,A -85,B 0,C 180,E1 162.066,E2 162.066} C_VEL
LIN {X 0,Y 752.257,Z 417.424,A -85,B 0,C 180,E1 159.417,E2 159.417} C_VEL
LIN {X 0,Y 752.379,Z 362.284,A -85,B 0,C 180,E1 156.586,E2 156.586} C_VEL
LIN {X 0,Y 752.492,Z 307.934,A -85,B 0,C 180,E1 153.738,E2 153.738} C_VEL
LIN {X 0,Y 752.583,Z 254.056,A -85,B 0,C 180,E1 150.86,E2 150.86} C_VEL
LIN {X 0,Y 752.671,Z 201.517,A -85,B 0,C 180,E1 147.991,E2 147.991} C_VEL
LIN {X 0,Y 752.478,Z 193.596,A -85,B 0,C 180,E1 147.542,E2 147.542} C_VEL
LIN {X 0,Y 751.962,Z 191.568,A -85,B 0,C 180,E1 147.393,E2 147.393} C_VEL
LIN {X 0,Y 751.971,Z 191.559,A -85,B 0,C 180,E1 144.466,E2 144.466} C_VEL
LIN {X 0,Y 751.922,Z 191.566,A -85,B 0,C 180,E1 141.681,E2 141.681} C_VEL
LIN {X 0,Y 751.926,Z 191.567,A -85,B 0,C 180,E1 139.053,E2 139.053} C_VEL
LIN {X 0,Y 751.942,Z 191.561,A -85,B 0,C 180,E1 136.114,E2 136.114} C_VEL
LIN {X 0,Y 751.958,Z 191.564,A -85,B 0,C 180,E1 133.325,E2 133.325} C_VEL
LIN {X 0,Y 751.97,Z 191.561,A -85,B 0,C 180,E1 130.458,E2 130.458} C_VEL
LIN {X 0,Y 751.896,Z 191.567,A -85,B 0,C 180,E1 127.618,E2 127.618} C_VEL
LIN {X 0,Y 751.975,Z 191.567,A -85,B 0,C 180,E1 124.966,E2 124.966} C_VEL
LIN {X 0,Y 751.989,Z 191.757,A -85,B 0,C 180,E1 123.036,E2 123.036} C_VEL
LIN {X 0,Y 752.683,Z 195.206,A -85,B 0,C 180,E1 122.764,E2 122.764} C_VEL
LIN {X 0,Y 752.559,Z 237.189,A -85,B 0,C 180,E1 119.932,E2 119.932} C_VEL
LIN {X 0,Y 752.445,Z 278.045,A -85,B 0,C 180,E1 117.251,E2 117.251} C_VEL
LIN {X 0,Y 752.489,Z 304.728,A -85,B 0,C 180,E1 115.556,E2 115.556} C_VEL
LIN {X 0,Y 752.564,Z 509.773,A -85,B 0,C 180,E1 113.446,E2 113.446} C_VEL
LIN {X 0,Y 752.502,Z 608.173,A -85,B 0,C 180,E1 112.427,E2 112.427} C_VEL
LIN {X 0,Y 752.467,Z 629.934,A -85,B 0,C 180,E1 112.061,E2 112.061} C_VEL
LIN {X 0,Y 752.401,Z 651.555,A -85,B 0,C 180,E1 111.558,E2 111.558} C_VEL
LIN {X 0,Y 752.359,Z 671.97,A -85,B 0,C 180,E1 110.947,E2 110.947} C_VEL
LIN {X 0,Y 752.31,Z 691.62,A -85,B 0,C 180,E1 110.216,E2 110.216} C_VEL
LIN {X 0,Y 752.24,Z 711.995,A -85,B 0,C 180,E1 109.309,E2 109.309} C_VEL
LIN {X 0,Y 752.189,Z 730.643,A -85,B 0,C 180,E1 108.324,E2 108.324} C_VEL
LIN {X 0,Y 752.124,Z 748.364,A -85,B 0,C 180,E1 107.22,E2 107.22} C_VEL
LIN {X 0,Y 752.075,Z 765.609,A -85,B 0,C 180,E1 105.975,E2 105.975} C_VEL
LIN {X 0,Y 752.023,Z 781.521,A -85,B 0,C 180,E1 104.633,E2 104.633} C_VEL
LIN {X 0,Y 751.987,Z 795.517,A -85,B 0,C 180,E1 103.265,E2 103.265} C_VEL
LIN {X 0,Y 751.957,Z 808.092,A -85,B 0,C 180,E1 101.816,E2 101.816} C_VEL
LIN {X 0,Y 751.943,Z 819.54,A -85,B 0,C 180,E1 100.258,E2 100.258} C_VEL
LIN {X 0,Y 751.927,Z 829.021,A -85,B 0,C 180,E1 98.719,E2 98.719} C_VEL
LIN {X 0,Y 751.923,Z 837.026,A -85,B 0,C 180,E1 97.104,E2 97.104} C_VEL
LIN {X 0,Y 751.912,Z 843.251,A -85,B 0,C 180,E1 95.494,E2 95.494} C_VEL
LIN {X 0,Y 751.914,Z 847.891,A -85,B 0,C 180,E1 93.889,E2 93.889} C_VEL
LIN {X 0,Y 751.91,Z 850.94,A -85,B 0,C 180,E1 92.21,E2 92.21} C_VEL
LIN {X 0,Y 751.9,Z 852.365,A -85,B 0,C 180,E1 90.457,E2 90.457} C_VEL
LIN {X 0,Y 751.9,Z 852.053,A -85,B 0,C 180,E1 88.781,E2 88.781} C_VEL
LIN {X 0,Y 751.911,Z 850.178,A -85,B 0,C 180,E1 87.18,E2 87.18} C_VEL
LIN {X 0,Y 751.916,Z 846.523,A -85,B 0,C 180,E1 85.5,E2 85.5} C_VEL
LIN {X 0,Y 751.922,Z 841.146,A -85,B 0,C 180,E1 83.817,E2 83.817} C_VEL
LIN {X 0,Y 751.908,Z 834.613,A -85,B 0,C 180,E1 82.281,E2 82.281} C_VEL
LIN {X 0,Y 751.919,Z 825.944,A -85,B 0,C 180,E1 80.663,E2 80.663} C_VEL
LIN {X 0,Y 751.938,Z 815.876,A -85,B 0,C 180,E1 79.116,E2 79.116} C_VEL
LIN {X 0,Y 751.963,Z 804.355,A -85,B 0,C 180,E1 77.638,E2 77.638} C_VEL
LIN {X 0,Y 751.993,Z 791.447,A -85,B 0,C 180,E1 76.231,E2 76.231} C_VEL
LIN {X 0,Y 752.036,Z 776.825,A -85,B 0,C 180,E1 74.858,E2 74.858} C_VEL
LIN {X 0,Y 752.09,Z 760.604,A -85,B 0,C 180,E1 73.55,E2 73.55} C_VEL
LIN {X 0,Y 752.135,Z 743.315,A -85,B 0,C 180,E1 72.356,E2 72.356} C_VEL
LIN {X 0,Y 752.198,Z 725.014,A -85,B 0,C 180,E1 71.275,E2 71.275} C_VEL
LIN {X 0,Y 752.267,Z 704.917,A -85,B 0,C 180,E1 70.269,E2 70.269} C_VEL
LIN {X 0,Y 752.326,Z 685.794,A -85,B 0,C 180,E1 69.459,E2 69.459} C_VEL
LIN {X 0,Y 752.379,Z 665.874,A -85,B 0,C 180,E1 68.768,E2 68.768} C_VEL
LIN {X 0,Y 752.43,Z 643.294,A -85,B 0,C 180,E1 68.143,E2 68.143} C_VEL
LIN {X 0,Y 752.476,Z 622.182,A -85,B 0,C 180,E1 67.7,E2 67.7} C_VEL
LIN {X 0,Y 752.51,Z 601.168,A -85,B 0,C 180,E1 67.399,E2 67.399} C_VEL
LIN {X 0,Y 752.676,Z 308.211,A -85,B 0,C 180,E1 64.397,E2 64.397} C_VEL
LIN {X 0,Y 752.398,Z 304.113,A -85,B 0,C 180,E1 64.338,E2 64.338} C_VEL
LIN {X 0,Y 752.519,Z 258.409,A -85,B 0,C 180,E1 61.38,E2 61.38} C_VEL
LIN {X 0,Y 752.608,Z 216.167,A -85,B 0,C 180,E1 58.57,E2 58.57} C_VEL
LIN {X 0,Y 752.567,Z 193.836,A -85,B 0,C 180,E1 57.046,E2 57.046} C_VEL
LIN {X 0,Y 751.936,Z 191.567,A -85,B 0,C 180,E1 56.848,E2 56.848} C_VEL
LIN {X 0,Y 751.967,Z 191.562,A -85,B 0,C 180,E1 54.076,E2 54.076} C_VEL
LIN {X 0,Y 751.945,Z 191.558,A -85,B 0,C 180,E1 51.222,E2 51.222} C_VEL
LIN {X 0,Y 751.976,Z 191.566,A -85,B 0,C 180,E1 48.33,E2 48.33} C_VEL
LIN {X 0,Y 751.962,Z 191.555,A -85,B 0,C 180,E1 45.349,E2 45.349} C_VEL
LIN {X 0,Y 751.969,Z 191.565,A -85,B 0,C 180,E1 42.389,E2 42.389} C_VEL
LIN {X 0,Y 751.967,Z 191.554,A -85,B 0,C 180,E1 39.366,E2 39.366} C_VEL
LIN {X 0,Y 751.971,Z 191.565,A -85,B 0,C 180,E1 36.374,E2 36.374} C_VEL
LIN {X 0,Y 751.975,Z 191.552,A -85,B 0,C 180,E1 33.31,E2 33.31} C_VEL
LIN {X 0,Y 751.978,Z 191.566,A -85,B 0,C 180,E1 30.262,E2 30.262} C_VEL
LIN {X 0,Y 751.971,Z 191.553,A -85,B 0,C 180,E1 27.221,E2 27.221} C_VEL
LIN {X 0,Y 751.973,Z 191.564,A -85,B 0,C 180,E1 24.193,E2 24.193} C_VEL
LIN {X 0,Y 751.976,Z 191.553,A -85,B 0,C 180,E1 21.203,E2 21.203} C_VEL
LIN {X 0,Y 751.976,Z 191.565,A -85,B 0,C 180,E1 18.209,E2 18.209} C_VEL
LIN {X 0,Y 751.979,Z 191.552,A -85,B 0,C 180,E1 15.186,E2 15.186} C_VEL
LIN {X 0,Y 751.97,Z 191.564,A -85,B 0,C 180,E1 12.128,E2 12.128} C_VEL
LIN {X 0,Y 751.977,Z 191.553,A -85,B 0,C 180,E1 9.104,E2 9.104} C_VEL
LIN {X 0,Y 751.971,Z 191.564,A -85,B 0,C 180,E1 6.106,E2 6.106} C_VEL
LIN {X 0,Y 751.968,Z 191.554,A -85,B 0,C 180,E1 3.125,E2 3.125} C_VEL
LIN {X 0,Y 751.969,Z 191.563,A -85,B 0,C 180,E1 0.076,E2 0.076} C_VEL
LIN {X 0,Y 751.964,Z 191.554,A -85,B 0,C 180,E1 -2.896,E2 -2.896} C_VEL
LIN {X 0,Y 751.966,Z 191.563,A -85,B 0,C 180,E1 -5.953,E2 -5.953} C_VEL
LIN {X 0,Y 751.947,Z 191.556,A -85,B 0,C 180,E1 -8.796,E2 -8.796} C_VEL
LIN {X 0,Y 751.972,Z 191.564,A -85,B 0,C 180,E1 -11.738,E2 -11.738} C_VEL
LIN {X 0,Y 751.933,Z 191.56,A -85,B 0,C 180,E1 -14.519,E2 -14.519} C_VEL
LIN {X 0,Y 751.973,Z 191.556,A -85,B 0,C 180,E1 -17.329,E2 -17.329} C_VEL
LIN {X 0,Y 751.942,Z 191.563,A -85,B 0,C 180,E1 -20.227,E2 -20.227} C_VEL
LIN {X 0,Y 751.949,Z 191.556,A -85,B 0,C 180,E1 -23.013,E2 -23.013} C_VEL
LIN {X 0,Y 751.963,Z 191.565,A -85,B 0,C 180,E1 -26.028,E2 -26.028} C_VEL
LIN {X 0,Y 751.927,Z 191.559,A -85,B 0,C 180,E1 -28.799,E2 -28.799} C_VEL
LIN {X 0,Y 751.972,Z 191.56,A -85,B 0,C 180,E1 -31.594,E2 -31.594} C_VEL
LIN {X 0,Y 751.927,Z 191.563,A -85,B 0,C 180,E1 -34.413,E2 -34.413} C_VEL
LIN {X 0,Y 751.936,Z 191.558,A -85,B 0,C 180,E1 -37.074,E2 -37.074} C_VEL
LIN {X 0,Y 751.963,Z 191.566,A -85,B 0,C 180,E1 -40.059,E2 -40.059} C_VEL
LIN {X 0,Y 751.915,Z 191.561,A -85,B 0,C 180,E1 -42.773,E2 -42.773} C_VEL
LIN {X 0,Y 751.975,Z 191.557,A -85,B 0,C 180,E1 -45.513,E2 -45.513} C_VEL
LIN {X 0,Y 751.923,Z 191.565,A -85,B 0,C 180,E1 -48.428,E2 -48.428} C_VEL
LIN {X 0,Y 751.912,Z 191.563,A -85,B 0,C 180,E1 -50.951,E2 -50.951} C_VEL
LIN {X 0,Y 751.997,Z 191.716,A -85,B 0,C 180,E1 -52.003,E2 -52.003} C_VEL
LIN {X 0,Y 753.176,Z 195.335,A -85,B 0,C 180,E1 -52.239,E2 -52.239} C_VEL
LIN {X 0,Y 753.045,Z 246.256,A -85,B 0,C 180,E1 -54.532,E2 -54.532} C_VEL
LIN {X 0,Y 753.039,Z 299.258,A -85,B 0,C 180,E1 -56.837,E2 -56.837} C_VEL
LIN {X 0,Y 753.011,Z 482.255,A -85,B 0,C 180,E1 -58.855,E2 -58.855} C_VEL
LIN {X 0,Y 752.88,Z 690.317,A -85,B 0,C 180,E1 -61.117,E2 -61.117} C_VEL
LIN {X 0,Y 752.816,Z 714.951,A -85,B 0,C 180,E1 -61.514,E2 -61.514} C_VEL
LIN {X 0,Y 752.759,Z 736.493,A -85,B 0,C 180,E1 -61.992,E2 -61.992} C_VEL
LIN {X 0,Y 752.689,Z 756.949,A -85,B 0,C 180,E1 -62.551,E2 -62.551} C_VEL
LIN {X 0,Y 752.615,Z 781.11,A -85,B 0,C 180,E1 -63.36,E2 -63.36} C_VEL
LIN {X 0,Y 752.545,Z 800.249,A -85,B 0,C 180,E1 -64.121,E2 -64.121} C_VEL
LIN {X 0,Y 752.468,Z 821.463,A -85,B 0,C 180,E1 -65.088,E2 -65.088} C_VEL
LIN {X 0,Y 752.363,Z 842.518,A -85,B 0,C 180,E1 -66.212,E2 -66.212} C_VEL
LIN {X 0,Y 752.295,Z 862.354,A -85,B 0,C 180,E1 -67.411,E2 -67.411} C_VEL
LIN {X 0,Y 752.197,Z 881.68,A -85,B 0,C 180,E1 -68.759,E2 -68.759} C_VEL
LIN {X 0,Y 752.125,Z 899.816,A -85,B 0,C 180,E1 -70.184,E2 -70.184} C_VEL
LIN {X 0,Y 752.084,Z 915.944,A -85,B 0,C 180,E1 -71.634,E2 -71.634} C_VEL
LIN {X 0,Y 752.014,Z 931.676,A -85,B 0,C 180,E1 -73.23,E2 -73.23} C_VEL
LIN {X 0,Y 751.976,Z 944.607,A -85,B 0,C 180,E1 -74.735,E2 -74.735} C_VEL
LIN {X 0,Y 751.965,Z 957.329,A -85,B 0,C 180,E1 -76.414,E2 -76.414} C_VEL
LIN {X 0,Y 751.937,Z 968.175,A -85,B 0,C 180,E1 -78.105,E2 -78.105} C_VEL
LIN {X 0,Y 751.937,Z 977.231,A -85,B 0,C 180,E1 -79.744,E2 -79.744} C_VEL
LIN {X 0,Y 751.902,Z 985.821,A -85,B 0,C 180,E1 -81.645,E2 -81.645} C_VEL
LIN {X 0,Y 751.91,Z 991.489,A -85,B 0,C 180,E1 -83.203,E2 -83.203} C_VEL
LIN {X 0,Y 751.888,Z 996.701,A -85,B 0,C 180,E1 -85.041,E2 -85.041} C_VEL
LIN {X 0,Y 751.892,Z 1000.009,A -85,B 0,C 180,E1 -86.798,E2 -86.798} C_VEL
LIN {X 0,Y 751.898,Z 1001.898,A -85,B 0,C 180,E1 -88.476,E2 -88.476} C_VEL
LIN {X 0,Y 751.885,Z 1002.395,A -85,B 0,C 180,E1 -90.381,E2 -90.381} C_VEL
LIN {X 0,Y 751.914,Z 1001.497,A -85,B 0,C 180,E1 -91.981,E2 -91.981} C_VEL
LIN {X 0,Y 751.913,Z 998.922,A -85,B 0,C 180,E1 -93.889,E2 -93.889} C_VEL
LIN {X 0,Y 751.904,Z 994.893,A -85,B 0,C 180,E1 -95.647,E2 -95.647} C_VEL
LIN {X 0,Y 751.888,Z 989.708,A -85,B 0,C 180,E1 -97.335,E2 -97.335} C_VEL
LIN {X 0,Y 751.923,Z 982.309,A -85,B 0,C 180,E1 -99.182,E2 -99.182} C_VEL
LIN {X 0,Y 751.909,Z 974.74,A -85,B 0,C 180,E1 -100.73,E2 -100.73} C_VEL
LIN {X 0,Y 751.955,Z 964.931,A -85,B 0,C 180,E1 -102.44,E2 -102.44} C_VEL
LIN {X 0,Y 751.978,Z 953.108,A -85,B 0,C 180,E1 -104.162,E2 -104.162} C_VEL
LIN {X 0,Y 752.003,Z 940.115,A -85,B 0,C 180,E1 -105.818,E2 -105.818} C_VEL
LIN {X 0,Y 752.047,Z 925.618,A -85,B 0,C 180,E1 -107.407,E2 -107.407} C_VEL
LIN {X 0,Y 752.093,Z 909.989,A -85,B 0,C 180,E1 -108.929,E2 -108.929} C_VEL
LIN {X 0,Y 752.164,Z 892.832,A -85,B 0,C 180,E1 -110.383,E2 -110.383} C_VEL
LIN {X 0,Y 752.239,Z 874.473,A -85,B 0,C 180,E1 -111.768,E2 -111.768} C_VEL
LIN {X 0,Y 752.311,Z 855.738,A -85,B 0,C 180,E1 -113.001,E2 -113.001} C_VEL
LIN {X 0,Y 752.413,Z 835.152,A -85,B 0,C 180,E1 -114.203,E2 -114.203} C_VEL
LIN {X 0,Y 752.488,Z 814.341,A -85,B 0,C 180,E1 -115.248,E2 -115.248} C_VEL
LIN {X 0,Y 752.568,Z 793.275,A -85,B 0,C 180,E1 -116.175,E2 -116.175} C_VEL
LIN {X 0,Y 752.643,Z 770.231,A -85,B 0,C 180,E1 -117.023,E2 -117.023} C_VEL
LIN {X 0,Y 752.711,Z 750.339,A -85,B 0,C 180,E1 -117.642,E2 -117.642} C_VEL
LIN {X 0,Y 752.794,Z 725.121,A -85,B 0,C 180,E1 -118.275,E2 -118.275} C_VEL
LIN {X 0,Y 752.853,Z 704.23,A -85,B 0,C 180,E1 -118.674,E2 -118.674} C_VEL
LIN {X 0,Y 752.883,Z 683.242,A -85,B 0,C 180,E1 -118.973,E2 -118.973} C_VEL
LIN {X 0,Y 753.026,Z 437.454,A -85,B 0,C 180,E1 -121.634,E2 -121.634} C_VEL
LIN {X 0,Y 753,Z 299.016,A -85,B 0,C 180,E1 -123.167,E2 -123.167} C_VEL
LIN {X 0,Y 753.055,Z 242.058,A -85,B 0,C 180,E1 -125.654,E2 -125.654} C_VEL
LIN {X 0,Y 753.192,Z 194.943,A -85,B 0,C 180,E1 -127.778,E2 -127.778} C_VEL
LIN {X 0,Y 751.954,Z 191.564,A -85,B 0,C 180,E1 -128.024,E2 -128.024} C_VEL
LIN {X 0,Y 751.93,Z 191.566,A -85,B 0,C 180,E1 -131.064,E2 -131.064} C_VEL
LIN {X 0,Y 751.937,Z 191.566,A -85,B 0,C 180,E1 -133.747,E2 -133.747} C_VEL
LIN {X 0,Y 751.965,Z 191.562,A -85,B 0,C 180,E1 -136.675,E2 -136.675} C_VEL
LIN {X 0,Y 751.927,Z 191.567,A -85,B 0,C 180,E1 -139.52,E2 -139.52} C_VEL
LIN {X 0,Y 751.97,Z 191.562,A -85,B 0,C 180,E1 -142.386,E2 -142.386} C_VEL
LIN {X 0,Y 751.926,Z 191.567,A -85,B 0,C 180,E1 -145.309,E2 -145.309} C_VEL
LIN {X 0,Y 752.003,Z 191.814,A -85,B 0,C 180,E1 -147.589,E2 -147.589} C_VEL
LIN {X 0,Y 752.705,Z 195.046,A -85,B 0,C 180,E1 -147.8,E2 -147.8} C_VEL
LIN {X 0,Y 752.544,Z 245.903,A -85,B 0,C 180,E1 -150.553,E2 -150.553} C_VEL
LIN {X 0,Y 752.472,Z 304.583,A -85,B 0,C 180,E1 -153.652,E2 -153.652} C_VEL
LIN {X 0,Y 752.372,Z 357.357,A -85,B 0,C 180,E1 -156.42,E2 -156.42} C_VEL
LIN {X 0,Y 752.253,Z 412.462,A -85,B 0,C 180,E1 -159.254,E2 -159.254} C_VEL
LIN {X 0,Y 752.142,Z 464.375,A -85,B 0,C 180,E1 -161.876,E2 -161.876} C_VEL
LIN {X 0,Y 752.211,Z 470.681,A -85,B 0,C 180,E1 -162.168,E2 -162.168} C_VEL
LIN {X 0,Y 752.205,Z 679.866,A -85,B 0,C 180,E1 -164.233,E2 -164.233} C_VEL
LIN {X 0,Y 752.179,Z 698.91,A -85,B 0,C 180,E1 -164.567,E2 -164.567} C_VEL
LIN {X 0,Y 752.151,Z 716.707,A -85,B 0,C 180,E1 -165.015,E2 -165.015} C_VEL
LIN {X 0,Y 752.094,Z 734.398,A -85,B 0,C 180,E1 -165.605,E2 -165.605} C_VEL
LIN {X 0,Y 752.083,Z 751.156,A -85,B 0,C 180,E1 -166.311,E2 -166.311} C_VEL
LIN {X 0,Y 752.047,Z 767.03,A -85,B 0,C 180,E1 -167.132,E2 -167.132} C_VEL
LIN {X 0,Y 752.014,Z 781.972,A -85,B 0,C 180,E1 -168.068,E2 -168.068} C_VEL
LIN {X 0,Y 751.983,Z 795.905,A -85,B 0,C 180,E1 -169.116,E2 -169.116} C_VEL
LIN {X 0,Y 751.959,Z 808.728,A -85,B 0,C 180,E1 -170.278,E2 -170.278} C_VEL
LIN {X 0,Y 751.939,Z 819.989,A -85,B 0,C 180,E1 -171.512,E2 -171.512} C_VEL
LIN {X 0,Y 751.93,Z 829.702,A -85,B 0,C 180,E1 -172.819,E2 -172.819} C_VEL
LIN {X 0,Y 751.919,Z 837.439,A -85,B 0,C 180,E1 -174.123,E2 -174.123} C_VEL
LIN {X 0,Y 751.912,Z 843.732,A -85,B 0,C 180,E1 -175.5,E2 -175.5} C_VEL
LIN {X 0,Y 751.916,Z 848.457,A -85,B 0,C 180,E1 -176.951,E2 -176.951} C_VEL
LIN {X 0,Y 751.91,Z 851.333,A -85,B 0,C 180,E1 -178.4,E2 -178.4} C_VEL
LIN {X 0,Y 751.911,Z 852.449,A -85,B 0,C 180,E1 -179.848,E2 -179.848} C_VEL
LIN {X 0,Y 751.915,Z 851.822,A -85,B 0,C 180,E1 -181.295,E2 -181.295} C_VEL
LIN {X 0,Y 751.911,Z 849.442,A -85,B 0,C 180,E1 -182.744,E2 -182.744} C_VEL
LIN {X 0,Y 751.913,Z 845.241,A -85,B 0,C 180,E1 -184.194,E2 -184.194} C_VEL
LIN {X 0,Y 751.92,Z 839.929,A -85,B 0,C 180,E1 -185.471,E2 -185.471} C_VEL
LIN {X 0,Y 750.931,Z 837.282,A -85,B 0,C 180,E1 -186.023,E2 -186.023} C_VEL
LIN {X 0,Y 745.826,Z 830.999,A -85,B 0,C 180,E1 -187.151,E2 -187.151} C_VEL
LIN {X 0,Y 744.047,Z 827.019,A -85,B 0,C 180,E1 -187.749,E2 -187.749} C_VEL
LIN {X 0,Y 743.951,Z 825.924,A -85,B 0,C 180,E1 -187.899,E2 -187.899} C_VEL
LIN {X 0,Y 743.984,Z 816.161,A -85,B 0,C 180,E1 -189.125,E2 -189.125} C_VEL
LIN {X 0,Y 744.022,Z 804.314,A -85,B 0,C 180,E1 -190.348,E2 -190.348} C_VEL
LIN {X 0,Y 744.075,Z 791.184,A -85,B 0,C 180,E1 -191.472,E2 -191.472} C_VEL
LIN {X 0,Y 744.139,Z 776.238,A -85,B 0,C 180,E1 -192.533,E2 -192.533} C_VEL
LIN {X 0,Y 744.21,Z 760.792,A -85,B 0,C 180,E1 -193.441,E2 -193.441} C_VEL
LIN {X 0,Y 744.268,Z 744.372,A -85,B 0,C 180,E1 -194.232,E2 -194.232} C_VEL
LIN {X 0,Y 744.343,Z 726.973,A -85,B 0,C 180,E1 -194.907,E2 -194.907} C_VEL
LIN {X 0,Y 744.425,Z 708.94,A -85,B 0,C 180,E1 -195.449,E2 -195.449} C_VEL
LIN {X 0,Y 744.47,Z 690.348,A -85,B 0,C 180,E1 -195.857,E2 -195.857} C_VEL
LIN {X 0,Y 744.511,Z 671.297,A -85,B 0,C 180,E1 -196.127,E2 -196.127} C_VEL
LIN {X 0,Y 744.485,Z 470.648,A -85,B 0,C 180,E1 -198.114,E2 -198.114} C_VEL
LIN {X 0,Y 744.625,Z 423.007,A -85,B 0,C 180,E1 -200.516,E2 -200.516} C_VEL
LIN {X 0,Y 744.817,Z 367.77,A -85,B 0,C 180,E1 -203.377,E2 -203.377} C_VEL
LIN {X 0,Y 745.023,Z 315.115,A -85,B 0,C 180,E1 -206.156,E2 -206.156} C_VEL
LIN {X 0,Y 745.23,Z 261.949,A -85,B 0,C 180,E1 -209.015,E2 -209.015} C_VEL
LIN {X 0,Y 745.483,Z 211.004,A -85,B 0,C 180,E1 -211.811,E2 -211.811} C_VEL
LIN {X 0,Y 745.406,Z 196.888,A -85,B 0,C 180,E1 -212.605,E2 -212.605} C_VEL
LIN {X 0,Y 744.033,Z 192.556,A -85,B 0,C 180,E1 -212.929,E2 -212.929} C_VEL
LIN {X 0,Y 744.026,Z 192.553,A -85,B 0,C 180,E1 -215.869,E2 -215.869} C_VEL
LIN {X 0,Y 743.972,Z 192.554,A -85,B 0,C 180,E1 -218.581,E2 -218.581} C_VEL
LIN {X 0,Y 744.042,Z 192.553,A -85,B 0,C 180,E1 -221.42,E2 -221.42} C_VEL
LIN {X 0,Y 744.001,Z 192.552,A -85,B 0,C 180,E1 -224.249,E2 -224.249} C_VEL
LIN {X 0,Y 744.008,Z 192.55,A -85,B 0,C 180,E1 -226.979,E2 -226.979} C_VEL
LIN {X 0,Y 744.038,Z 192.555,A -85,B 0,C 180,E1 -229.877,E2 -229.877} C_VEL
LIN {X 0,Y 743.96,Z 192.557,A -85,B 0,C 180,E1 -232.591,E2 -232.591} C_VEL
LIN {X 0,Y 744.033,Z 192.553,A -85,B 0,C 180,E1 -235.332,E2 -235.332} C_VEL
LIN {X 0,Y 744.058,Z 192.756,A -85,B 0,C 180,E1 -236.635,E2 -236.635} C_VEL
LIN {X 0,Y 745.472,Z 197.7,A -85,B 0,C 180,E1 -237.051,E2 -237.051} C_VEL
LIN {X 0,Y 745.224,Z 239.994,A -85,B 0,C 180,E1 -239.931,E2 -239.931} C_VEL
LIN {X 0,Y 744.994,Z 280.787,A -85,B 0,C 180,E1 -242.633,E2 -242.633} C_VEL
LIN {X 0,Y 744.954,Z 304.588,A -85,B 0,C 180,E1 -244.164,E2 -244.164} C_VEL
LIN {X 0,Y 745.451,Z 308.865,A -85,B 0,C 180,E1 -244.228,E2 -244.228} C_VEL
LIN {X 0,Y 745.108,Z 606.026,A -85,B 0,C 180,E1 -247.311,E2 -247.311} C_VEL
LIN {X 0,Y 745.032,Z 628.423,A -85,B 0,C 180,E1 -247.676,E2 -247.676} C_VEL
LIN {X 0,Y 744.911,Z 650.851,A -85,B 0,C 180,E1 -248.194,E2 -248.194} C_VEL
LIN {X 0,Y 744.834,Z 670.731,A -85,B 0,C 180,E1 -248.79,E2 -248.79} C_VEL
LIN {X 0,Y 744.711,Z 690.941,A -85,B 0,C 180,E1 -249.539,E2 -249.539} C_VEL
LIN {X 0,Y 744.589,Z 710.755,A -85,B 0,C 180,E1 -250.421,E2 -250.421} C_VEL
LIN {X 0,Y 744.477,Z 729.942,A -85,B 0,C 180,E1 -251.439,E2 -251.439} C_VEL
LIN {X 0,Y 744.344,Z 747.092,A -85,B 0,C 180,E1 -252.508,E2 -252.508} C_VEL
LIN {X 0,Y 744.238,Z 764.104,A -85,B 0,C 180,E1 -253.732,E2 -253.732} C_VEL
LIN {X 0,Y 744.149,Z 779.82,A -85,B 0,C 180,E1 -255.049,E2 -255.049} C_VEL
LIN {X 0,Y 744.08,Z 793.662,A -85,B 0,C 180,E1 -256.399,E2 -256.399} C_VEL
LIN {X 0,Y 744.023,Z 806.182,A -85,B 0,C 180,E1 -257.819,E2 -257.819} C_VEL
LIN {X 0,Y 743.968,Z 817.952,A -85,B 0,C 180,E1 -259.39,E2 -259.39} C_VEL
LIN {X 0,Y 743.938,Z 827.717,A -85,B 0,C 180,E1 -260.952,E2 -260.952} C_VEL
LIN {X 0,Y 743.914,Z 835.617,A -85,B 0,C 180,E1 -262.509,E2 -262.509} C_VEL
LIN {X 0,Y 743.913,Z 842.243,A -85,B 0,C 180,E1 -264.137,E2 -264.137} C_VEL
LIN {X 0,Y 743.918,Z 847.31,A -85,B 0,C 180,E1 -265.838,E2 -265.838} C_VEL
LIN {X 0,Y 743.912,Z 850.605,A -85,B 0,C 180,E1 -267.535,E2 -267.535} C_VEL
LIN {X 0,Y 743.913,Z 852.279,A -85,B 0,C 180,E1 -269.23,E2 -269.23} C_VEL
LIN {X 0,Y 743.912,Z 852.232,A -85,B 0,C 180,E1 -271.001,E2 -271.001} C_VEL
LIN {X 0,Y 743.913,Z 850.512,A -85,B 0,C 180,E1 -272.619,E2 -272.619} C_VEL
LIN {X 0,Y 743.917,Z 846.935,A -85,B 0,C 180,E1 -274.394,E2 -274.394} C_VEL
LIN {X 0,Y 743.924,Z 841.747,A -85,B 0,C 180,E1 -276.095,E2 -276.095} C_VEL
LIN {X 0,Y 743.916,Z 834.966,A -85,B 0,C 180,E1 -277.724,E2 -277.724} C_VEL
LIN {X 0,Y 743.937,Z 826.406,A -85,B 0,C 180,E1 -279.36,E2 -279.36} C_VEL
LIN {X 0,Y 743.975,Z 816.449,A -85,B 0,C 180,E1 -280.924,E2 -280.924} C_VEL
LIN {X 0,Y 744.019,Z 804.355,A -85,B 0,C 180,E1 -282.496,E2 -282.496} C_VEL
LIN {X 0,Y 744.08,Z 791.443,A -85,B 0,C 180,E1 -283.918,E2 -283.918} C_VEL
LIN {X 0,Y 744.166,Z 777.258,A -85,B 0,C 180,E1 -285.269,E2 -285.269} C_VEL
LIN {X 0,Y 744.266,Z 761.395,A -85,B 0,C 180,E1 -286.568,E2 -286.568} C_VEL
LIN {X 0,Y 744.357,Z 744.516,A -85,B 0,C 180,E1 -287.754,E2 -287.754} C_VEL
LIN {X 0,Y 744.485,Z 726.467,A -85,B 0,C 180,E1 -288.845,E2 -288.845} C_VEL
LIN {X 0,Y 744.621,Z 706.683,A -85,B 0,C 180,E1 -289.861,E2 -289.861} C_VEL
LIN {X 0,Y 744.729,Z 687.838,A -85,B 0,C 180,E1 -290.678,E2 -290.678} C_VEL
LIN {X 0,Y 744.846,Z 668.001,A -85,B 0,C 180,E1 -291.388,E2 -291.388} C_VEL
LIN {X 0,Y 744.956,Z 646.302,A -85,B 0,C 180,E1 -292.015,E2 -292.015} C_VEL
LIN {X 0,Y 745.044,Z 624.296,A -85,B 0,C 180,E1 -292.496,E2 -292.496} C_VEL
LIN {X 0,Y 745.114,Z 603.079,A -85,B 0,C 180,E1 -292.815,E2 -292.815} C_VEL
LIN {X 0,Y 745.454,Z 308.627,A -85,B 0,C 180,E1 -295.865,E2 -295.865} C_VEL
LIN {X 0,Y 744.892,Z 304.088,A -85,B 0,C 180,E1 -295.941,E2 -295.941} C_VEL
LIN {X 0,Y 745.133,Z 259.06,A -85,B 0,C 180,E1 -298.887,E2 -298.887} C_VEL
LIN {X 0,Y 745.348,Z 216.751,A -85,B 0,C 180,E1 -301.732,E2 -301.732} C_VEL
LIN {X 0,Y 745.365,Z 197.018,A -85,B 0,C 180,E1 -303.092,E2 -303.092} C_VEL
LIN {X 0,Y 744.02,Z 192.557,A -85,B 0,C 180,E1 -303.482,E2 -303.482} C_VEL
LIN {X 0,Y 744.024,Z 192.545,A -85,B 0,C 180,E1 -306.537,E2 -306.537} C_VEL
LIN {X 0,Y 744.013,Z 192.554,A -85,B 0,C 180,E1 -309.398,E2 -309.398} C_VEL
LIN {X 0,Y 744.03,Z 192.545,A -85,B 0,C 180,E1 -312.342,E2 -312.342} C_VEL
LIN {X 0,Y 744.002,Z 192.55,A -85,B 0,C 180,E1 -315.124,E2 -315.124} C_VEL
LIN {X 0,Y 744.028,Z 192.553,A -85,B 0,C 180,E1 -317.887,E2 -317.887} C_VEL
LIN {X 0,Y 744.024,Z 192.544,A -85,B 0,C 180,E1 -320.73,E2 -320.73} C_VEL
LIN {X 0,Y 744.035,Z 192.553,A -85,B 0,C 180,E1 -323.655,E2 -323.655} C_VEL
LIN {X 0,Y 744.033,Z 192.541,A -85,B 0,C 180,E1 -326.709,E2 -326.709} C_VEL
LIN {X 0,Y 744.039,Z 192.555,A -85,B 0,C 180,E1 -329.738,E2 -329.738} C_VEL
LIN {X 0,Y 744.033,Z 192.542,A -85,B 0,C 180,E1 -332.725,E2 -332.725} C_VEL
LIN {X 0,Y 744.035,Z 192.554,A -85,B 0,C 180,E1 -335.718,E2 -335.718} C_VEL
LIN {X 0,Y 744.037,Z 192.542,A -85,B 0,C 180,E1 -338.807,E2 -338.807} C_VEL
LIN {X 0,Y 744.033,Z 192.552,A -85,B 0,C 180,E1 -341.833,E2 -341.833} C_VEL
LIN {X 0,Y 744.035,Z 192.542,A -85,B 0,C 180,E1 -344.888,E2 -344.888} C_VEL
LIN {X 0,Y 744.029,Z 192.552,A -85,B 0,C 180,E1 -347.898,E2 -347.898} C_VEL
LIN {X 0,Y 744.037,Z 192.542,A -85,B 0,C 180,E1 -350.876,E2 -350.876} C_VEL
LIN {X 0,Y 744.03,Z 192.552,A -85,B 0,C 180,E1 -353.906,E2 -353.906} C_VEL
LIN {X 0,Y 744.032,Z 192.543,A -85,B 0,C 180,E1 -356.919,E2 -356.919} C_VEL
LIN {X 0,Y 744.03,Z 192.551,A -85,B 0,C 180,E1 -359.923,E2 -359.923} C_VEL
LIN {X 0,Y 744.021,Z 192.543,A -85,B 0,C 180,E1 -362.85,E2 -362.85} C_VEL
LIN {X 0,Y 744.032,Z 192.553,A -85,B 0,C 180,E1 -365.862,E2 -365.862} C_VEL
LIN {X 0,Y 744.004,Z 192.545,A -85,B 0,C 180,E1 -368.735,E2 -368.735} C_VEL
LIN {X 0,Y 744.029,Z 192.551,A -85,B 0,C 180,E1 -371.63,E2 -371.63} C_VEL
LIN {X 0,Y 743.996,Z 192.55,A -85,B 0,C 180,E1 -374.397,E2 -374.397} C_VEL
LIN {X 0,Y 744.037,Z 192.543,A -85,B 0,C 180,E1 -377.197,E2 -377.197} C_VEL
LIN {X 0,Y 744.005,Z 192.552,A -85,B 0,C 180,E1 -380.206,E2 -380.206} C_VEL
LIN {X 0,Y 744.011,Z 192.545,A -85,B 0,C 180,E1 -383.022,E2 -383.022} C_VEL
LIN {X 0,Y 744.02,Z 192.553,A -85,B 0,C 180,E1 -386.069,E2 -386.069} C_VEL
LIN {X 0,Y 743.991,Z 192.547,A -85,B 0,C 180,E1 -388.848,E2 -388.848} C_VEL
LIN {X 0,Y 744.034,Z 192.551,A -85,B 0,C 180,E1 -391.715,E2 -391.715} C_VEL
LIN {X 0,Y 743.984,Z 192.551,A -85,B 0,C 180,E1 -394.528,E2 -394.528} C_VEL
LIN {X 0,Y 744.012,Z 192.546,A -85,B 0,C 180,E1 -397.212,E2 -397.212} C_VEL
LIN {X 0,Y 743.998,Z 192.554,A -85,B 0,C 180,E1 -400.274,E2 -400.274} C_VEL
LIN {X 0,Y 743.982,Z 192.549,A -85,B 0,C 180,E1 -402.953,E2 -402.953} C_VEL
LIN {X 0,Y 744.037,Z 192.552,A -85,B 0,C 180,E1 -405.776,E2 -405.776} C_VEL
LIN {X 0,Y 743.975,Z 192.553,A -85,B 0,C 180,E1 -408.605,E2 -408.605} C_VEL
LIN {X 0,Y 743.992,Z 192.552,A -85,B 0,C 180,E1 -411.215,E2 -411.215} C_VEL
LIN {X 0,Y 744.057,Z 192.701,A -85,B 0,C 180,E1 -411.57,E2 -411.57} C_VEL
LIN {X 0,Y 745.441,Z 196.178,A -85,B 0,C 180,E1 -411.816,E2 -411.816} C_VEL
LIN {X 0,Y 746.508,Z 198.953,A -85,B 0,C 180,E1 -412.009,E2 -412.009} C_VEL
LIN {X 0,Y 746.231,Z 250.452,A -85,B 0,C 180,E1 -414.348,E2 -414.348} C_VEL
LIN {X 0,Y 746.107,Z 299.285,A -85,B 0,C 180,E1 -416.489,E2 -416.489} C_VEL
LIN {X 0,Y 746.45,Z 304.512,A -85,B 0,C 180,E1 -416.566,E2 -416.566} C_VEL
LIN {X 0,Y 746.056,Z 566.743,A -85,B 0,C 180,E1 -419.462,E2 -419.462} C_VEL
LIN {X 0,Y 745.863,Z 690.638,A -85,B 0,C 180,E1 -420.823,E2 -420.823} C_VEL
LIN {X 0,Y 745.738,Z 715.738,A -85,B 0,C 180,E1 -421.235,E2 -421.235} C_VEL
LIN {X 0,Y 745.629,Z 737.035,A -85,B 0,C 180,E1 -421.714,E2 -421.714} C_VEL
LIN {X 0,Y 745.494,Z 759.081,A -85,B 0,C 180,E1 -422.326,E2 -422.326} C_VEL
LIN {X 0,Y 745.323,Z 782.798,A -85,B 0,C 180,E1 -423.143,E2 -423.143} C_VEL
LIN {X 0,Y 745.177,Z 803.236,A -85,B 0,C 180,E1 -423.974,E2 -423.974} C_VEL
LIN {X 0,Y 744.963,Z 826.334,A -85,B 0,C 180,E1 -425.074,E2 -425.074} C_VEL
LIN {X 0,Y 744.817,Z 845.357,A -85,B 0,C 180,E1 -426.12,E2 -426.12} C_VEL
LIN {X 0,Y 744.621,Z 867.232,A -85,B 0,C 180,E1 -427.499,E2 -427.499} C_VEL
LIN {X 0,Y 744.486,Z 884.825,A -85,B 0,C 180,E1 -428.763,E2 -428.763} C_VEL
LIN {X 0,Y 744.329,Z 902.603,A -85,B 0,C 180,E1 -430.213,E2 -430.213} C_VEL
LIN {X 0,Y 744.248,Z 918.496,A -85,B 0,C 180,E1 -431.677,E2 -431.677} C_VEL
LIN {X 0,Y 744.132,Z 933.8,A -85,B 0,C 180,E1 -433.289,E2 -433.289} C_VEL
LIN {X 0,Y 744.053,Z 946.534,A -85,B 0,C 180,E1 -434.808,E2 -434.808} C_VEL
LIN {X 0,Y 743.994,Z 959.233,A -85,B 0,C 180,E1 -436.556,E2 -436.556} C_VEL
LIN {X 0,Y 743.968,Z 968.782,A -85,B 0,C 180,E1 -438.079,E2 -438.079} C_VEL
LIN {X 0,Y 743.952,Z 978.399,A -85,B 0,C 180,E1 -439.859,E2 -439.859} C_VEL
LIN {X 0,Y 743.91,Z 986.206,A -85,B 0,C 180,E1 -441.653,E2 -441.653} C_VEL
LIN {X 0,Y 743.909,Z 991.997,A -85,B 0,C 180,E1 -443.285,E2 -443.285} C_VEL
LIN {X 0,Y 743.902,Z 997.178,A -85,B 0,C 180,E1 -445.22,E2 -445.22} C_VEL
LIN {X 0,Y 743.89,Z 1000.122,A -85,B 0,C 180,E1 -446.841,E2 -446.841} C_VEL
LIN {X 0,Y 743.902,Z 1002.032,A -85,B 0,C 180,E1 -448.614,E2 -448.614} C_VEL
LIN {X 0,Y 743.883,Z 1002.373,A -85,B 0,C 180,E1 -450.462,E2 -450.462} C_VEL
LIN {X 0,Y 743.916,Z 1001.43,A -85,B 0,C 180,E1 -452.08,E2 -452.08} C_VEL
LIN {X 0,Y 743.916,Z 998.605,A -85,B 0,C 180,E1 -454.085,E2 -454.085} C_VEL
LIN {X 0,Y 743.919,Z 994.687,A -85,B 0,C 180,E1 -455.786,E2 -455.786} C_VEL
LIN {X 0,Y 743.893,Z 988.936,A -85,B 0,C 180,E1 -457.647,E2 -457.647} C_VEL
LIN {X 0,Y 743.929,Z 981.6,A -85,B 0,C 180,E1 -459.438,E2 -459.438} C_VEL
LIN {X 0,Y 743.926,Z 973.925,A -85,B 0,C 180,E1 -461.003,E2 -461.003} C_VEL
LIN {X 0,Y 743.978,Z 962.87,A -85,B 0,C 180,E1 -462.891,E2 -462.891} C_VEL
LIN {X 0,Y 744.04,Z 952.531,A -85,B 0,C 180,E1 -464.396,E2 -464.396} C_VEL
LIN {X 0,Y 744.114,Z 939.175,A -85,B 0,C 180,E1 -466.101,E2 -466.101} C_VEL
LIN {X 0,Y 744.189,Z 924.842,A -85,B 0,C 180,E1 -467.677,E2 -467.677} C_VEL
LIN {X 0,Y 744.313,Z 909.099,A -85,B 0,C 180,E1 -469.216,E2 -469.216} C_VEL
LIN {X 0,Y 744.42,Z 892.325,A -85,B 0,C 180,E1 -470.646,E2 -470.646} C_VEL
LIN {X 0,Y 744.581,Z 873.871,A -85,B 0,C 180,E1 -472.045,E2 -472.045} C_VEL
LIN {X 0,Y 744.718,Z 854.774,A -85,B 0,C 180,E1 -473.311,E2 -473.311} C_VEL
LIN {X 0,Y 744.932,Z 833.551,A -85,B 0,C 180,E1 -474.546,E2 -474.546} C_VEL
LIN {X 0,Y 745.075,Z 813.454,A -85,B 0,C 180,E1 -475.56,E2 -475.56} C_VEL
LIN {X 0,Y 745.289,Z 791.18,A -85,B 0,C 180,E1 -476.536,E2 -476.536} C_VEL
LIN {X 0,Y 745.407,Z 768.835,A -85,B 0,C 180,E1 -477.355,E2 -477.355} C_VEL
LIN {X 0,Y 745.561,Z 747.322,A -85,B 0,C 180,E1 -478.019,E2 -478.019} C_VEL
LIN {X 0,Y 745.712,Z 723.126,A -85,B 0,C 180,E1 -478.611,E2 -478.611} C_VEL
LIN {X 0,Y 745.811,Z 702.773,A -85,B 0,C 180,E1 -478.995,E2 -478.995} C_VEL
LIN {X 0,Y 745.891,Z 678.577,A -85,B 0,C 180,E1 -479.329,E2 -479.329} C_VEL
LIN {X 0,Y 746.202,Z 441.144,A -85,B 0,C 180,E1 -481.917,E2 -481.917} C_VEL
LIN {X 0,Y 746.303,Z 300.452,A -85,B 0,C 180,E1 -483.488,E2 -483.488} C_VEL
LIN {X 0,Y 746.003,Z 297.647,A -85,B 0,C 180,E1 -483.565,E2 -483.565} C_VEL
LIN {X 0,Y 746.291,Z 239.96,A -85,B 0,C 180,E1 -486.123,E2 -486.123} C_VEL
LIN {X 0,Y 746.493,Z 198.687,A -85,B 0,C 180,E1 -488.004,E2 -488.004} C_VEL
LIN {X 0,Y 744.077,Z 192.825,A -85,B 0,C 180,E1 -488.423,E2 -488.423} C_VEL
LIN {X 0,Y 744.039,Z 192.553,A -85,B 0,C 180,E1 -488.576,E2 -488.576} C_VEL
LIN {X 0,Y 744.001,Z 192.556,A -85,B 0,C 180,E1 -491.416,E2 -491.416} C_VEL
LIN {X 0,Y 744.014,Z 192.553,A -85,B 0,C 180,E1 -494.249,E2 -494.249} C_VEL
LIN {X 0,Y 744.012,Z 192.553,A -85,B 0,C 180,E1 -497.154,E2 -497.154} C_VEL
LIN {X 0,Y 743.983,Z 192.556,A -85,B 0,C 180,E1 -499.826,E2 -499.826} C_VEL
LIN {X 0,Y 744.027,Z 192.551,A -85,B 0,C 180,E1 -502.838,E2 -502.838} C_VEL
LIN {X 0,Y 743.984,Z 192.557,A -85,B 0,C 180,E1 -505.635,E2 -505.635} C_VEL
LIN {X 0,Y 744.038,Z 192.756,A -85,B 0,C 180,E1 -507.254,E2 -507.254} C_VEL
LIN {X 0,Y 745.545,Z 197.578,A -85,B 0,C 180,E1 -507.602,E2 -507.602} C_VEL
LIN {X 0,Y 745.188,Z 248.742,A -85,B 0,C 180,E1 -510.41,E2 -510.41} C_VEL
LIN {X 0,Y 744.994,Z 307.417,A -85,B 0,C 180,E1 -513.539,E2 -513.539} C_VEL
LIN {X 0,Y 744.851,Z 358.166,A -85,B 0,C 180,E1 -516.209,E2 -516.209} C_VEL
LIN {X 0,Y 744.628,Z 413.271,A -85,B 0,C 180,E1 -519.072,E2 -519.072} C_VEL
LIN {X 0,Y 744.433,Z 464.385,A -85,B 0,C 180,E1 -521.681,E2 -521.681} C_VEL
LIN {X 0,Y 744.488,Z 470.658,A -85,B 0,C 180,E1 -521.976,E2 -521.976} C_VEL
LIN {X 0,Y 744.501,Z 679.899,A -85,B 0,C 180,E1 -524.066,E2 -524.066} C_VEL
LIN {X 0,Y 744.452,Z 699.025,A -85,B 0,C 180,E1 -524.405,E2 -524.405} C_VEL
LIN {X 0,Y 744.396,Z 716.721,A -85,B 0,C 180,E1 -524.855,E2 -524.855} C_VEL
LIN {X 0,Y 744.305,Z 734.408,A -85,B 0,C 180,E1 -525.451,E2 -525.451} C_VEL
LIN {X 0,Y 744.258,Z 751.163,A -85,B 0,C 180,E1 -526.164,E2 -526.164} C_VEL
LIN {X 0,Y 744.185,Z 767.034,A -85,B 0,C 180,E1 -526.994,E2 -526.994} C_VEL
LIN {X 0,Y 744.115,Z 781.977,A -85,B 0,C 180,E1 -527.939,E2 -527.939} C_VEL
LIN {X 0,Y 744.052,Z 795.91,A -85,B 0,C 180,E1 -528.999,E2 -528.999} C_VEL
LIN {X 0,Y 744.004,Z 808.735,A -85,B 0,C 180,E1 -530.173,E2 -530.173} C_VEL
LIN {X 0,Y 743.967,Z 819.994,A -85,B 0,C 180,E1 -531.42,E2 -531.42} C_VEL
LIN {X 0,Y 743.941,Z 829.706,A -85,B 0,C 180,E1 -532.742,E2 -532.742} C_VEL
LIN {X 0,Y 743.927,Z 837.442,A -85,B 0,C 180,E1 -534.06,E2 -534.06} C_VEL
LIN {X 0,Y 743.914,Z 843.735,A -85,B 0,C 180,E1 -535.452,E2 -535.452} C_VEL
LIN {X 0,Y 743.915,Z 848.459,A -85,B 0,C 180,E1 -536.918,E2 -536.918} C_VEL
LIN {X 0,Y 743.91,Z 851.335,A -85,B 0,C 180,E1 -538.383,E2 -538.383} C_VEL
LIN {X 0,Y 743.912,Z 852.449,A -85,B 0,C 180,E1 -539.846,E2 -539.846} C_VEL
LIN {X 0,Y 743.915,Z 851.822,A -85,B 0,C 180,E1 -541.309,E2 -541.309} C_VEL
LIN {X 0,Y 743.911,Z 849.441,A -85,B 0,C 180,E1 -542.774,E2 -542.774} C_VEL
LIN {X 0,Y 743.916,Z 845.239,A -85,B 0,C 180,E1 -544.239,E2 -544.239} C_VEL
LIN {X 0,Y 743.922,Z 839.468,A -85,B 0,C 180,E1 -545.631,E2 -545.631} C_VEL
LIN {X 0,Y 743.938,Z 831.809,A -85,B 0,C 180,E1 -547.025,E2 -547.025} C_VEL
LIN {X 0,Y 743.951,Z 825.924,A -85,B 0,C 180,E1 -547.899,E2 -547.899} C_VEL
LIN {X 0,Y 742.947,Z 822.182,A -85,B 0,C 180,E1 -548.413,E2 -548.413} C_VEL
LIN {X 0,Y 736.999,Z 811.994,A -85,B 0,C 180,E1 -549.678,E2 -549.678} C_VEL
LIN {X 0,Y 736.061,Z 807.368,A -85,B 0,C 180,E1 -550.165,E2 -550.165} C_VEL
LIN {X 0,Y 736.147,Z 794.187,A -85,B 0,C 180,E1 -551.359,E2 -551.359} C_VEL
LIN {X 0,Y 736.239,Z 780.45,A -85,B 0,C 180,E1 -552.391,E2 -552.391} C_VEL
LIN {X 0,Y 736.345,Z 765.149,A -85,B 0,C 180,E1 -553.347,E2 -553.347} C_VEL
LIN {X 0,Y 736.456,Z 748.826,A -85,B 0,C 180,E1 -554.186,E2 -554.186} C_VEL
LIN {X 0,Y 736.543,Z 732.574,A -85,B 0,C 180,E1 -554.867,E2 -554.867} C_VEL
LIN {X 0,Y 736.667,Z 715.014,A -85,B 0,C 180,E1 -555.449,E2 -555.449} C_VEL
LIN {X 0,Y 736.748,Z 696.185,A -85,B 0,C 180,E1 -555.914,E2 -555.914} C_VEL
LIN {X 0,Y 736.815,Z 677.437,A -85,B 0,C 180,E1 -556.228,E2 -556.228} C_VEL
LIN {X 0,Y 736.875,Z 471.438,A -85,B 0,C 180,E1 -558.299,E2 -558.299} C_VEL
LIN {X 0,Y 736.706,Z 469.344,A -85,B 0,C 180,E1 -558.354,E2 -558.354} C_VEL
LIN {X 0,Y 736.999,Z 417.464,A -85,B 0,C 180,E1 -561.026,E2 -561.026} C_VEL
LIN {X 0,Y 737.322,Z 362.245,A -85,B 0,C 180,E1 -563.921,E2 -563.921} C_VEL
LIN {X 0,Y 737.639,Z 309.296,A -85,B 0,C 180,E1 -566.746,E2 -566.746} C_VEL
LIN {X 0,Y 737.969,Z 256.1,A -85,B 0,C 180,E1 -569.64,E2 -569.64} C_VEL
LIN {X 0,Y 738.306,Z 205.365,A -85,B 0,C 180,E1 -572.464,E2 -572.464} C_VEL
LIN {X 0,Y 738.149,Z 199.426,A -85,B 0,C 180,E1 -572.809,E2 -572.809} C_VEL
LIN {X 0,Y 736.097,Z 193.541,A -85,B 0,C 180,E1 -573.249,E2 -573.249} C_VEL
LIN {X 0,Y 736.091,Z 193.54,A -85,B 0,C 180,E1 -576.221,E2 -576.221} C_VEL
LIN {X 0,Y 736.047,Z 193.543,A -85,B 0,C 180,E1 -579.01,E2 -579.01} C_VEL
LIN {X 0,Y 736.041,Z 193.543,A -85,B 0,C 180,E1 -582.005,E2 -582.005} C_VEL
LIN {X 0,Y 736.098,Z 193.543,A -85,B 0,C 180,E1 -584.73,E2 -584.73} C_VEL
LIN {X 0,Y 736.095,Z 193.538,A -85,B 0,C 180,E1 -587.748,E2 -587.748} C_VEL
LIN {X 0,Y 736.025,Z 193.544,A -85,B 0,C 180,E1 -590.522,E2 -590.522} C_VEL
LIN {X 0,Y 736.094,Z 193.545,A -85,B 0,C 180,E1 -593.296,E2 -593.296} C_VEL
LIN {X 0,Y 736.07,Z 193.543,A -85,B 0,C 180,E1 -596.238,E2 -596.238} C_VEL
LIN {X 0,Y 736.099,Z 193.755,A -85,B 0,C 180,E1 -596.297,E2 -596.297} C_VEL
LIN {X 0,Y 738.265,Z 201.005,A -85,B 0,C 180,E1 -596.92,E2 -596.92} C_VEL
LIN {X 0,Y 737.884,Z 244.526,A -85,B 0,C 180,E1 -599.909,E2 -599.909} C_VEL
LIN {X 0,Y 737.524,Z 286.731,A -85,B 0,C 180,E1 -602.726,E2 -602.726} C_VEL
LIN {X 0,Y 737.486,Z 304.705,A -85,B 0,C 180,E1 -603.884,E2 -603.884} C_VEL
LIN {X 0,Y 738.246,Z 309.769,A -85,B 0,C 180,E1 -603.966,E2 -603.966} C_VEL
LIN {X 0,Y 737.722,Z 605.718,A -85,B 0,C 180,E1 -607.067,E2 -607.067} C_VEL
LIN {X 0,Y 737.611,Z 628.128,A -85,B 0,C 180,E1 -607.432,E2 -607.432} C_VEL
LIN {X 0,Y 737.451,Z 650.107,A -85,B 0,C 180,E1 -607.94,E2 -607.94} C_VEL
LIN {X 0,Y 737.311,Z 670.74,A -85,B 0,C 180,E1 -608.563,E2 -608.563} C_VEL
LIN {X 0,Y 737.125,Z 690.777,A -85,B 0,C 180,E1 -609.311,E2 -609.311} C_VEL
LIN {X 0,Y 736.946,Z 710.839,A -85,B 0,C 180,E1 -610.213,E2 -610.213} C_VEL
LIN {X 0,Y 736.764,Z 729.945,A -85,B 0,C 180,E1 -611.238,E2 -611.238} C_VEL
LIN {X 0,Y 736.568,Z 747.698,A -85,B 0,C 180,E1 -612.358,E2 -612.358} C_VEL
LIN {X 0,Y 736.398,Z 765.633,A -85,B 0,C 180,E1 -613.676,E2 -613.676} C_VEL
LIN {X 0,Y 736.255,Z 781.529,A -85,B 0,C 180,E1 -615.046,E2 -615.046} C_VEL
LIN {X 0,Y 736.161,Z 795.183,A -85,B 0,C 180,E1 -616.41,E2 -616.41} C_VEL
LIN {X 0,Y 736.072,Z 808.109,A -85,B 0,C 180,E1 -617.925,E2 -617.925} C_VEL
LIN {X 0,Y 736.001,Z 819.508,A -85,B 0,C 180,E1 -619.511,E2 -619.511} C_VEL
LIN {X 0,Y 735.958,Z 829.031,A -85,B 0,C 180,E1 -621.09,E2 -621.09} C_VEL
LIN {X 0,Y 735.929,Z 837.035,A -85,B 0,C 180,E1 -622.741,E2 -622.741} C_VEL
LIN {X 0,Y 735.915,Z 843.511,A -85,B 0,C 180,E1 -624.464,E2 -624.464} C_VEL
LIN {X 0,Y 735.914,Z 848.226,A -85,B 0,C 180,E1 -626.183,E2 -626.183} C_VEL
LIN {X 0,Y 735.913,Z 851.164,A -85,B 0,C 180,E1 -627.898,E2 -627.898} C_VEL
LIN {X 0,Y 735.9,Z 852.393,A -85,B 0,C 180,E1 -629.611,E2 -629.611} C_VEL
LIN {X 0,Y 735.897,Z 851.985,A -85,B 0,C 180,E1 -631.324,E2 -631.324} C_VEL
LIN {X 0,Y 735.902,Z 850.057,A -85,B 0,C 180,E1 -632.96,E2 -632.96} C_VEL
LIN {X 0,Y 735.909,Z 846.323,A -85,B 0,C 180,E1 -634.676,E2 -634.676} C_VEL
LIN {X 0,Y 735.923,Z 840.836,A -85,B 0,C 180,E1 -636.397,E2 -636.397} C_VEL
LIN {X 0,Y 735.938,Z 834.257,A -85,B 0,C 180,E1 -637.966,E2 -637.966} C_VEL
LIN {X 0,Y 735.962,Z 825.945,A -85,B 0,C 180,E1 -639.541,E2 -639.541} C_VEL
LIN {X 0,Y 736.015,Z 815.869,A -85,B 0,C 180,E1 -641.123,E2 -641.123} C_VEL
LIN {X 0,Y 736.084,Z 804.355,A -85,B 0,C 180,E1 -642.633,E2 -642.633} C_VEL
LIN {X 0,Y 736.171,Z 791.44,A -85,B 0,C 180,E1 -644.071,E2 -644.071} C_VEL
LIN {X 0,Y 736.309,Z 776.329,A -85,B 0,C 180,E1 -645.517,E2 -645.517} C_VEL
LIN {X 0,Y 736.462,Z 760.328,A -85,B 0,C 180,E1 -646.828,E2 -646.828} C_VEL
LIN {X 0,Y 736.609,Z 743.893,A -85,B 0,C 180,E1 -647.988,E2 -647.988} C_VEL
LIN {X 0,Y 736.785,Z 725.738,A -85,B 0,C 180,E1 -649.09,E2 -649.09} C_VEL
LIN {X 0,Y 736.991,Z 705.777,A -85,B 0,C 180,E1 -650.116,E2 -650.116} C_VEL
LIN {X 0,Y 737.168,Z 686.768,A -85,B 0,C 180,E1 -650.941,E2 -650.941} C_VEL
LIN {X 0,Y 737.336,Z 667.135,A -85,B 0,C 180,E1 -651.645,E2 -651.645} C_VEL
LIN {X 0,Y 737.509,Z 644.02,A -85,B 0,C 180,E1 -652.305,E2 -652.305} C_VEL
LIN {X 0,Y 737.632,Z 623.057,A -85,B 0,C 180,E1 -652.755,E2 -652.755} C_VEL
LIN {X 0,Y 737.732,Z 602.367,A -85,B 0,C 180,E1 -653.064,E2 -653.064} C_VEL
LIN {X 0,Y 738.247,Z 309.8,A -85,B 0,C 180,E1 -656.123,E2 -656.123} C_VEL
LIN {X 0,Y 737.404,Z 304.095,A -85,B 0,C 180,E1 -656.223,E2 -656.223} C_VEL
LIN {X 0,Y 737.753,Z 260.372,A -85,B 0,C 180,E1 -659.115,E2 -659.115} C_VEL
LIN {X 0,Y 738.089,Z 218.791,A -85,B 0,C 180,E1 -661.939,E2 -661.939} C_VEL
LIN {X 0,Y 738.056,Z 199.649,A -85,B 0,C 180,E1 -663.276,E2 -663.276} C_VEL
LIN {X 0,Y 736.094,Z 193.544,A -85,B 0,C 180,E1 -663.809,E2 -663.809} C_VEL
LIN {X 0,Y 736.069,Z 193.537,A -85,B 0,C 180,E1 -666.729,E2 -666.729} C_VEL
LIN {X 0,Y 736.092,Z 193.545,A -85,B 0,C 180,E1 -669.628,E2 -669.628} C_VEL
LIN {X 0,Y 736.08,Z 193.534,A -85,B 0,C 180,E1 -672.675,E2 -672.675} C_VEL
LIN {X 0,Y 736.092,Z 193.545,A -85,B 0,C 180,E1 -675.608,E2 -675.608} C_VEL
LIN {X 0,Y 736.086,Z 193.533,A -85,B 0,C 180,E1 -678.693,E2 -678.693} C_VEL
LIN {X 0,Y 736.09,Z 193.544,A -85,B 0,C 180,E1 -681.627,E2 -681.627} C_VEL
LIN {X 0,Y 736.09,Z 193.532,A -85,B 0,C 180,E1 -684.725,E2 -684.725} C_VEL
LIN {X 0,Y 736.095,Z 193.542,A -85,B 0,C 180,E1 -687.735,E2 -687.735} C_VEL
LIN {X 0,Y 736.097,Z 193.53,A -85,B 0,C 180,E1 -690.724,E2 -690.724} C_VEL
LIN {X 0,Y 736.095,Z 193.544,A -85,B 0,C 180,E1 -693.715,E2 -693.715} C_VEL
LIN {X 0,Y 736.095,Z 193.528,A -85,B 0,C 180,E1 -696.801,E2 -696.801} C_VEL
LIN {X 0,Y 736.095,Z 193.542,A -85,B 0,C 180,E1 -699.823,E2 -699.823} C_VEL
LIN {X 0,Y 736.097,Z 193.529,A -85,B 0,C 180,E1 -702.856,E2 -702.856} C_VEL
LIN {X 0,Y 736.091,Z 193.54,A -85,B 0,C 180,E1 -705.903,E2 -705.903} C_VEL
LIN {X 0,Y 736.097,Z 193.529,A -85,B 0,C 180,E1 -708.879,E2 -708.879} C_VEL
LIN {X 0,Y 736.093,Z 193.542,A -85,B 0,C 180,E1 -711.879,E2 -711.879} C_VEL
LIN {X 0,Y 736.092,Z 193.529,A -85,B 0,C 180,E1 -714.856,E2 -714.856} C_VEL
LIN {X 0,Y 736.092,Z 193.543,A -85,B 0,C 180,E1 -717.898,E2 -717.898} C_VEL
LIN {X 0,Y 736.094,Z 193.527,A -85,B 0,C 180,E1 -720.934,E2 -720.934} C_VEL
LIN {X 0,Y 736.085,Z 193.543,A -85,B 0,C 180,E1 -723.973,E2 -723.973} C_VEL
LIN {X 0,Y 736.085,Z 193.528,A -85,B 0,C 180,E1 -726.944,E2 -726.944} C_VEL
LIN {X 0,Y 736.083,Z 193.543,A -85,B 0,C 180,E1 -730.013,E2 -730.013} C_VEL
LIN {X 0,Y 736.079,Z 193.533,A -85,B 0,C 180,E1 -732.952,E2 -732.952} C_VEL
LIN {X 0,Y 736.083,Z 193.544,A -85,B 0,C 180,E1 -736.007,E2 -736.007} C_VEL
LIN {X 0,Y 736.064,Z 193.535,A -85,B 0,C 180,E1 -738.863,E2 -738.863} C_VEL
LIN {X 0,Y 736.095,Z 193.543,A -85,B 0,C 180,E1 -741.851,E2 -741.851} C_VEL
LIN {X 0,Y 736.05,Z 193.538,A -85,B 0,C 180,E1 -744.659,E2 -744.659} C_VEL
LIN {X 0,Y 736.094,Z 193.536,A -85,B 0,C 180,E1 -747.506,E2 -747.506} C_VEL
LIN {X 0,Y 736.053,Z 193.541,A -85,B 0,C 180,E1 -750.389,E2 -750.389} C_VEL
LIN {X 0,Y 736.067,Z 193.536,A -85,B 0,C 180,E1 -753.099,E2 -753.099} C_VEL
LIN {X 0,Y 736.066,Z 193.543,A -85,B 0,C 180,E1 -756.205,E2 -756.205} C_VEL
LIN {X 0,Y 736.045,Z 193.538,A -85,B 0,C 180,E1 -758.886,E2 -758.886} C_VEL
LIN {X 0,Y 736.097,Z 193.54,A -85,B 0,C 180,E1 -761.729,E2 -761.729} C_VEL
LIN {X 0,Y 736.042,Z 193.542,A -85,B 0,C 180,E1 -764.505,E2 -764.505} C_VEL
LIN {X 0,Y 736.049,Z 193.54,A -85,B 0,C 180,E1 -767.111,E2 -767.111} C_VEL
LIN {X 0,Y 736.078,Z 193.541,A -85,B 0,C 180,E1 -770.13,E2 -770.13} C_VEL
LIN {X 0,Y 736.048,Z 193.566,A -85,B 0,C 180,E1 -771.114,E2 -771.114} C_VEL
LIN {X 0,Y 737.361,Z 197.003,A -85,B 0,C 180,E1 -771.36,E2 -771.36} C_VEL
LIN {X 0,Y 739.844,Z 202.205,A -85,B 0,C 180,E1 -771.758,E2 -771.758} C_VEL
LIN {X 0,Y 739.438,Z 252.549,A -85,B 0,C 180,E1 -774.065,E2 -774.065} C_VEL
LIN {X 0,Y 739.213,Z 299.377,A -85,B 0,C 180,E1 -776.136,E2 -776.136} C_VEL
LIN {X 0,Y 739.767,Z 304.649,A -85,B 0,C 180,E1 -776.225,E2 -776.225} C_VEL
LIN {X 0,Y 739.162,Z 566.234,A -85,B 0,C 180,E1 -779.14,E2 -779.14} C_VEL
LIN {X 0,Y 738.866,Z 690.746,A -85,B 0,C 180,E1 -780.521,E2 -780.521} C_VEL
LIN {X 0,Y 738.682,Z 715.989,A -85,B 0,C 180,E1 -780.939,E2 -780.939} C_VEL
LIN {X 0,Y 738.517,Z 737.469,A -85,B 0,C 180,E1 -781.427,E2 -781.427} C_VEL
LIN {X 0,Y 738.315,Z 760.62,A -85,B 0,C 180,E1 -782.08,E2 -782.08} C_VEL
LIN {X 0,Y 738.046,Z 783.535,A -85,B 0,C 180,E1 -782.885,E2 -782.885} C_VEL
LIN {X 0,Y 737.827,Z 804.234,A -85,B 0,C 180,E1 -783.739,E2 -783.739} C_VEL
LIN {X 0,Y 737.502,Z 827.14,A -85,B 0,C 180,E1 -784.847,E2 -784.847} C_VEL
LIN {X 0,Y 737.279,Z 846.887,A -85,B 0,C 180,E1 -785.95,E2 -785.95} C_VEL
LIN {X 0,Y 736.994,Z 867.234,A -85,B 0,C 180,E1 -787.253,E2 -787.253} C_VEL
LIN {X 0,Y 736.79,Z 885.106,A -85,B 0,C 180,E1 -788.551,E2 -788.551} C_VEL
LIN {X 0,Y 736.562,Z 902.604,A -85,B 0,C 180,E1 -789.996,E2 -789.996} C_VEL
LIN {X 0,Y 736.424,Z 918.494,A -85,B 0,C 180,E1 -791.475,E2 -791.475} C_VEL
LIN {X 0,Y 736.241,Z 933.802,A -85,B 0,C 180,E1 -793.104,E2 -793.104} C_VEL
LIN {X 0,Y 736.14,Z 946.535,A -85,B 0,C 180,E1 -794.641,E2 -794.641} C_VEL
LIN {X 0,Y 736.044,Z 959.754,A -85,B 0,C 180,E1 -796.488,E2 -796.488} C_VEL
LIN {X 0,Y 736,Z 969.102,A -85,B 0,C 180,E1 -798.003,E2 -798.003} C_VEL
LIN {X 0,Y 735.967,Z 978.76,A -85,B 0,C 180,E1 -799.827,E2 -799.827} C_VEL
LIN {X 0,Y 735.912,Z 986.207,A -85,B 0,C 180,E1 -801.562,E2 -801.562} C_VEL
LIN {X 0,Y 735.917,Z 991.998,A -85,B 0,C 180,E1 -803.211,E2 -803.211} C_VEL
LIN {X 0,Y 735.898,Z 997.178,A -85,B 0,C 180,E1 -805.168,E2 -805.168} C_VEL
LIN {X 0,Y 735.892,Z 1000.122,A -85,B 0,C 180,E1 -806.807,E2 -806.807} C_VEL
LIN {X 0,Y 735.905,Z 1002.099,A -85,B 0,C 180,E1 -808.677,E2 -808.677} C_VEL
LIN {X 0,Y 735.881,Z 1002.351,A -85,B 0,C 180,E1 -810.545,E2 -810.545} C_VEL
LIN {X 0,Y 735.917,Z 1001.297,A -85,B 0,C 180,E1 -812.258,E2 -812.258} C_VEL
LIN {X 0,Y 735.914,Z 998.431,A -85,B 0,C 180,E1 -814.215,E2 -814.215} C_VEL
LIN {X 0,Y 735.923,Z 994.481,A -85,B 0,C 180,E1 -815.927,E2 -815.927} C_VEL
LIN {X 0,Y 735.907,Z 988.636,A -85,B 0,C 180,E1 -817.809,E2 -817.809} C_VEL
LIN {X 0,Y 735.937,Z 981.601,A -85,B 0,C 180,E1 -819.541,E2 -819.541} C_VEL
LIN {X 0,Y 735.951,Z 973.926,A -85,B 0,C 180,E1 -821.124,E2 -821.124} C_VEL
LIN {X 0,Y 736.02,Z 962.872,A -85,B 0,C 180,E1 -823.033,E2 -823.033} C_VEL
LIN {X 0,Y 736.106,Z 952.533,A -85,B 0,C 180,E1 -824.554,E2 -824.554} C_VEL
LIN {X 0,Y 736.223,Z 939.445,A -85,B 0,C 180,E1 -826.247,E2 -826.247} C_VEL
LIN {X 0,Y 736.329,Z 924.844,A -85,B 0,C 180,E1 -827.872,E2 -827.872} C_VEL
LIN {X 0,Y 736.525,Z 909.098,A -85,B 0,C 180,E1 -829.427,E2 -829.427} C_VEL
LIN {X 0,Y 736.688,Z 892.324,A -85,B 0,C 180,E1 -830.872,E2 -830.872} C_VEL
LIN {X 0,Y 736.935,Z 873.997,A -85,B 0,C 180,E1 -832.278,E2 -832.278} C_VEL
LIN {X 0,Y 737.141,Z 855.082,A -85,B 0,C 180,E1 -833.545,E2 -833.545} C_VEL
LIN {X 0,Y 737.455,Z 834.357,A -85,B 0,C 180,E1 -834.769,E2 -834.769} C_VEL
LIN {X 0,Y 737.671,Z 814.349,A -85,B 0,C 180,E1 -835.792,E2 -835.792} C_VEL
LIN {X 0,Y 737.994,Z 791.916,A -85,B 0,C 180,E1 -836.79,E2 -836.79} C_VEL
LIN {X 0,Y 738.186,Z 769.577,A -85,B 0,C 180,E1 -837.62,E2 -837.62} C_VEL
LIN {X 0,Y 738.413,Z 748.132,A -85,B 0,C 180,E1 -838.29,E2 -838.29} C_VEL
LIN {X 0,Y 738.644,Z 723.518,A -85,B 0,C 180,E1 -838.902,E2 -838.902} C_VEL
LIN {X 0,Y 738.787,Z 702.774,A -85,B 0,C 180,E1 -839.298,E2 -839.298} C_VEL
LIN {X 0,Y 738.912,Z 678.196,A -85,B 0,C 180,E1 -839.637,E2 -839.637} C_VEL
LIN {X 0,Y 739.404,Z 441.272,A -85,B 0,C 180,E1 -842.244,E2 -842.244} C_VEL
LIN {X 0,Y 739.616,Z 301.831,A -85,B 0,C 180,E1 -843.815,E2 -843.815} C_VEL
LIN {X 0,Y 739.094,Z 298.171,A -85,B 0,C 180,E1 -843.898,E2 -843.898} C_VEL
LIN {X 0,Y 739.553,Z 239.96,A -85,B 0,C 180,E1 -846.505,E2 -846.505} C_VEL
LIN {X 0,Y 739.783,Z 202.044,A -85,B 0,C 180,E1 -848.253,E2 -848.253} C_VEL
LIN {X 0,Y 736.248,Z 194.372,A -85,B 0,C 180,E1 -848.835,E2 -848.835} C_VEL
LIN {X 0,Y 736.098,Z 193.545,A -85,B 0,C 180,E1 -848.89,E2 -848.89} C_VEL
LIN {X 0,Y 736.098,Z 193.544,A -85,B 0,C 180,E1 -851.833,E2 -851.833} C_VEL
LIN {X 0,Y 736.094,Z 193.545,A -85,B 0,C 180,E1 -854.73,E2 -854.73} C_VEL
LIN {X 0,Y 736.094,Z 193.544,A -85,B 0,C 180,E1 -857.643,E2 -857.643} C_VEL
LIN {X 0,Y 736.1,Z 193.544,A -85,B 0,C 180,E1 -860.527,E2 -860.527} C_VEL
LIN {X 0,Y 736.087,Z 193.545,A -85,B 0,C 180,E1 -863.489,E2 -863.489} C_VEL
LIN {X 0,Y 736.101,Z 193.544,A -85,B 0,C 180,E1 -866.437,E2 -866.437} C_VEL
LIN {X 0,Y 736.114,Z 193.791,A -85,B 0,C 180,E1 -866.903,E2 -866.903} C_VEL
LIN {X 0,Y 738.426,Z 200.857,A -85,B 0,C 180,E1 -867.435,E2 -867.435} C_VEL
LIN {X 0,Y 737.861,Z 251.699,A -85,B 0,C 180,E1 -870.266,E2 -870.266} C_VEL
LIN {X 0,Y 737.516,Z 310.25,A -85,B 0,C 180,E1 -873.423,E2 -873.423} C_VEL
LIN {X 0,Y 737.327,Z 364.464,A -85,B 0,C 180,E1 -876.287,E2 -876.287} C_VEL
LIN {X 0,Y 736.992,Z 419.67,A -85,B 0,C 180,E1 -879.178,E2 -879.178} C_VEL
LIN {X 0,Y 736.751,Z 470.465,A -85,B 0,C 180,E1 -881.778,E2 -881.778} C_VEL
LIN {X 0,Y 737.012,Z 488.726,A -85,B 0,C 180,E1 -881.968,E2 -881.968} C_VEL
LIN {X 0,Y 736.806,Z 679.936,A -85,B 0,C 180,E1 -883.895,E2 -883.895} C_VEL
LIN {X 0,Y 736.732,Z 698.968,A -85,B 0,C 180,E1 -884.235,E2 -884.235} C_VEL
LIN {X 0,Y 736.649,Z 716.735,A -85,B 0,C 180,E1 -884.692,E2 -884.692} C_VEL
LIN {X 0,Y 736.523,Z 734.417,A -85,B 0,C 180,E1 -885.293,E2 -885.293} C_VEL
LIN {X 0,Y 736.439,Z 751.17,A -85,B 0,C 180,E1 -886.014,E2 -886.014} C_VEL
LIN {X 0,Y 736.329,Z 766.972,A -85,B 0,C 180,E1 -886.849,E2 -886.849} C_VEL
LIN {X 0,Y 736.223,Z 781.982,A -85,B 0,C 180,E1 -887.808,E2 -887.808} C_VEL
LIN {X 0,Y 736.125,Z 795.916,A -85,B 0,C 180,E1 -888.879,E2 -888.879} C_VEL
LIN {X 0,Y 736.049,Z 808.741,A -85,B 0,C 180,E1 -890.065,E2 -890.065} C_VEL
LIN {X 0,Y 735.996,Z 819.999,A -85,B 0,C 180,E1 -891.327,E2 -891.327} C_VEL
LIN {X 0,Y 735.954,Z 829.711,A -85,B 0,C 180,E1 -892.663,E2 -892.663} C_VEL
LIN {X 0,Y 735.933,Z 837.547,A -85,B 0,C 180,E1 -894.015,E2 -894.015} C_VEL
LIN {X 0,Y 735.917,Z 843.738,A -85,B 0,C 180,E1 -895.402,E2 -895.402} C_VEL
LIN {X 0,Y 735.915,Z 848.461,A -85,B 0,C 180,E1 -896.885,E2 -896.885} C_VEL
LIN {X 0,Y 735.911,Z 851.337,A -85,B 0,C 180,E1 -898.365,E2 -898.365} C_VEL
LIN {X 0,Y 735.912,Z 852.449,A -85,B 0,C 180,E1 -899.844,E2 -899.844} C_VEL
LIN {X 0,Y 735.914,Z 851.821,A -85,B 0,C 180,E1 -901.324,E2 -901.324} C_VEL
LIN {X 0,Y 735.912,Z 849.439,A -85,B 0,C 180,E1 -902.804,E2 -902.804} C_VEL
LIN {X 0,Y 735.919,Z 845.237,A -85,B 0,C 180,E1 -904.286,E2 -904.286} C_VEL
LIN {X 0,Y 735.926,Z 839.466,A -85,B 0,C 180,E1 -905.692,E2 -905.692} C_VEL
LIN {X 0,Y 735.954,Z 831.807,A -85,B 0,C 180,E1 -907.102,E2 -907.102} C_VEL
LIN {X 0,Y 735.986,Z 822.611,A -85,B 0,C 180,E1 -908.437,E2 -908.437} C_VEL
LIN {X 0,Y 736.04,Z 811.927,A -85,B 0,C 180,E1 -909.698,E2 -909.698} C_VEL
LIN {X 0,Y 736.061,Z 807.368,A -85,B 0,C 180,E1 -910.165,E2 -910.165} C_VEL
LIN {X 0,Y 735.127,Z 802.66,A -85,B 0,C 180,E1 -910.64,E2 -910.64} C_VEL
LIN {X 0,Y 729.255,Z 790.206,A -85,B 0,C 180,E1 -911.791,E2 -911.791} C_VEL
LIN {X 0,Y 728.304,Z 784.724,A -85,B 0,C 180,E1 -912.218,E2 -912.218} C_VEL
LIN {X 0,Y 728.445,Z 769.201,A -85,B 0,C 180,E1 -913.252,E2 -913.252} C_VEL
LIN {X 0,Y 728.599,Z 752.979,A -85,B 0,C 180,E1 -914.139,E2 -914.139} C_VEL
LIN {X 0,Y 728.729,Z 735.644,A -85,B 0,C 180,E1 -914.908,E2 -914.908} C_VEL
LIN {X 0,Y 728.892,Z 718.299,A -85,B 0,C 180,E1 -915.516,E2 -915.516} C_VEL
LIN {X 0,Y 729.006,Z 699.867,A -85,B 0,C 180,E1 -916.006,E2 -916.006} C_VEL
LIN {X 0,Y 729.105,Z 681.174,A -85,B 0,C 180,E1 -916.351,E2 -916.351} C_VEL
LIN {X 0,Y 729.162,Z 642.014,A -85,B 0,C 180,E1 -916.772,E2 -916.772} C_VEL
LIN {X 0,Y 729.244,Z 472.056,A -85,B 0,C 180,E1 -918.491,E2 -918.491} C_VEL
LIN {X 0,Y 729.002,Z 469.734,A -85,B 0,C 180,E1 -918.534,E2 -918.534} C_VEL
LIN {X 0,Y 729.384,Z 418.134,A -85,B 0,C 180,E1 -921.221,E2 -921.221} C_VEL
LIN {X 0,Y 729.793,Z 363.729,A -85,B 0,C 180,E1 -924.098,E2 -924.098} C_VEL
LIN {X 0,Y 730.225,Z 310.78,A -85,B 0,C 180,E1 -926.952,E2 -926.952} C_VEL
LIN {X 0,Y 730.682,Z 257.539,A -85,B 0,C 180,E1 -929.875,E2 -929.875} C_VEL
LIN {X 0,Y 731.155,Z 206.399,A -85,B 0,C 180,E1 -932.749,E2 -932.749} C_VEL
LIN {X 0,Y 731.053,Z 202.8,A -85,B 0,C 180,E1 -932.961,E2 -932.961} C_VEL
LIN {X 0,Y 728.145,Z 194.532,A -85,B 0,C 180,E1 -933.601,E2 -933.601} C_VEL
LIN {X 0,Y 728.129,Z 194.531,A -85,B 0,C 180,E1 -936.485,E2 -936.485} C_VEL
LIN {X 0,Y 728.137,Z 194.532,A -85,B 0,C 180,E1 -939.276,E2 -939.276} C_VEL
LIN {X 0,Y 728.098,Z 194.532,A -85,B 0,C 180,E1 -942.134,E2 -942.134} C_VEL
LIN {X 0,Y 728.153,Z 194.531,A -85,B 0,C 180,E1 -944.896,E2 -944.896} C_VEL
LIN {X 0,Y 728.154,Z 194.529,A -85,B 0,C 180,E1 -947.861,E2 -947.861} C_VEL
LIN {X 0,Y 728.083,Z 194.533,A -85,B 0,C 180,E1 -950.619,E2 -950.619} C_VEL
LIN {X 0,Y 728.161,Z 194.533,A -85,B 0,C 180,E1 -953.447,E2 -953.447} C_VEL
LIN {X 0,Y 728.144,Z 194.584,A -85,B 0,C 180,E1 -955.952,E2 -955.952} C_VEL
LIN {X 0,Y 731.081,Z 203.706,A -85,B 0,C 180,E1 -956.74,E2 -956.74} C_VEL
LIN {X 0,Y 730.554,Z 247.173,A -85,B 0,C 180,E1 -959.757,E2 -959.757} C_VEL
LIN {X 0,Y 730.071,Z 290.037,A -85,B 0,C 180,E1 -962.645,E2 -962.645} C_VEL
LIN {X 0,Y 730.002,Z 304.646,A -85,B 0,C 180,E1 -963.594,E2 -963.594} C_VEL
LIN {X 0,Y 731.053,Z 311.118,A -85,B 0,C 180,E1 -963.705,E2 -963.705} C_VEL
LIN {X 0,Y 730.351,Z 605.307,A -85,B 0,C 180,E1 -966.817,E2 -966.817} C_VEL
LIN {X 0,Y 730.203,Z 627.683,A -85,B 0,C 180,E1 -967.18,E2 -967.18} C_VEL
LIN {X 0,Y 729.999,Z 650.119,A -85,B 0,C 180,E1 -967.703,E2 -967.703} C_VEL
LIN {X 0,Y 729.8,Z 670.734,A -85,B 0,C 180,E1 -968.331,E2 -968.331} C_VEL
LIN {X 0,Y 729.555,Z 690.687,A -85,B 0,C 180,E1 -969.082,E2 -969.082} C_VEL
LIN {X 0,Y 729.297,Z 711.654,A -85,B 0,C 180,E1 -970.039,E2 -970.039} C_VEL
LIN {X 0,Y 729.049,Z 730.631,A -85,B 0,C 180,E1 -971.073,E2 -971.073} C_VEL
LIN {X 0,Y 728.799,Z 748.01,A -85,B 0,C 180,E1 -972.185,E2 -972.185} C_VEL
LIN {X 0,Y 728.575,Z 765.645,A -85,B 0,C 180,E1 -973.496,E2 -973.496} C_VEL
LIN {X 0,Y 728.381,Z 781.531,A -85,B 0,C 180,E1 -974.881,E2 -974.881} C_VEL
LIN {X 0,Y 728.245,Z 795.18,A -85,B 0,C 180,E1 -976.259,E2 -976.259} C_VEL
LIN {X 0,Y 728.128,Z 808.117,A -85,B 0,C 180,E1 -977.791,E2 -977.791} C_VEL
LIN {X 0,Y 728.028,Z 819.511,A -85,B 0,C 180,E1 -979.395,E2 -979.395} C_VEL
LIN {X 0,Y 727.971,Z 828.845,A -85,B 0,C 180,E1 -980.958,E2 -980.958} C_VEL
LIN {X 0,Y 727.933,Z 836.92,A -85,B 0,C 180,E1 -982.634,E2 -982.634} C_VEL
LIN {X 0,Y 727.914,Z 843.261,A -85,B 0,C 180,E1 -984.324,E2 -984.324} C_VEL
LIN {X 0,Y 727.918,Z 847.875,A -85,B 0,C 180,E1 -985.983,E2 -985.983} C_VEL
LIN {X 0,Y 727.91,Z 850.83,A -85,B 0,C 180,E1 -987.638,E2 -987.638} C_VEL
LIN {X 0,Y 727.903,Z 852.352,A -85,B 0,C 180,E1 -989.449,E2 -989.449} C_VEL
LIN {X 0,Y 727.902,Z 852.106,A -85,B 0,C 180,E1 -991.181,E2 -991.181} C_VEL
LIN {X 0,Y 727.909,Z 850.288,A -85,B 0,C 180,E1 -992.834,E2 -992.834} C_VEL
LIN {X 0,Y 727.916,Z 846.735,A -85,B 0,C 180,E1 -994.57,E2 -994.57} C_VEL
LIN {X 0,Y 727.932,Z 841.437,A -85,B 0,C 180,E1 -996.309,E2 -996.309} C_VEL
LIN {X 0,Y 727.947,Z 834.613,A -85,B 0,C 180,E1 -997.974,E2 -997.974} C_VEL
LIN {X 0,Y 727.987,Z 825.946,A -85,B 0,C 180,E1 -999.646,E2 -999.646} C_VEL
LIN {X 0,Y 728.064,Z 815.288,A -85,B 0,C 180,E1 -1001.326,E2 -1001.326} C_VEL
LIN {X 0,Y 728.162,Z 803.686,A -85,B 0,C 180,E1 -1002.853,E2 -1002.853} C_VEL
LIN {X 0,Y 728.281,Z 790.661,A -85,B 0,C 180,E1 -1004.308,E2 -1004.308} C_VEL
LIN {X 0,Y 728.457,Z 775.036,A -85,B 0,C 180,E1 -1005.802,E2 -1005.802} C_VEL
LIN {X 0,Y 728.66,Z 758.929,A -85,B 0,C 180,E1 -1007.118,E2 -1007.118} C_VEL
LIN {X 0,Y 728.895,Z 742.043,A -85,B 0,C 180,E1 -1008.309,E2 -1008.309} C_VEL
LIN {X 0,Y 729.168,Z 722.09,A -85,B 0,C 180,E1 -1009.506,E2 -1009.506} C_VEL
LIN {X 0,Y 729.388,Z 703.091,A -85,B 0,C 180,E1 -1010.461,E2 -1010.461} C_VEL
LIN {X 0,Y 729.656,Z 683.618,A -85,B 0,C 180,E1 -1011.293,E2 -1011.293} C_VEL
LIN {X 0,Y 729.908,Z 661.286,A -85,B 0,C 180,E1 -1012.067,E2 -1012.067} C_VEL
LIN {X 0,Y 730.093,Z 640.176,A -85,B 0,C 180,E1 -1012.637,E2 -1012.637} C_VEL
LIN {X 0,Y 730.285,Z 617.845,A -85,B 0,C 180,E1 -1013.089,E2 -1013.089} C_VEL
LIN {X 0,Y 730.4,Z 592.796,A -85,B 0,C 180,E1 -1013.42,E2 -1013.42} C_VEL
LIN {X 0,Y 731.059,Z 309.801,A -85,B 0,C 180,E1 -1016.399,E2 -1016.399} C_VEL
LIN {X 0,Y 729.935,Z 303.922,A -85,B 0,C 180,E1 -1016.524,E2 -1016.524} C_VEL
LIN {X 0,Y 730.388,Z 261.023,A -85,B 0,C 180,E1 -1019.392,E2 -1019.392} C_VEL
LIN {X 0,Y 730.864,Z 219.442,A -85,B 0,C 180,E1 -1022.246,E2 -1022.246} C_VEL
LIN {X 0,Y 730.869,Z 202.718,A -85,B 0,C 180,E1 -1023.432,E2 -1023.432} C_VEL
LIN {X 0,Y 728.154,Z 194.53,A -85,B 0,C 180,E1 -1024.169,E2 -1024.169} C_VEL
LIN {X 0,Y 728.122,Z 194.529,A -85,B 0,C 180,E1 -1026.976,E2 -1026.976} C_VEL
LIN {X 0,Y 728.157,Z 194.532,A -85,B 0,C 180,E1 -1029.785,E2 -1029.785} C_VEL
LIN {X 0,Y 728.138,Z 194.524,A -85,B 0,C 180,E1 -1032.72,E2 -1032.72} C_VEL
LIN {X 0,Y 728.156,Z 194.532,A -85,B 0,C 180,E1 -1035.678,E2 -1035.678} C_VEL
LIN {X 0,Y 728.148,Z 194.522,A -85,B 0,C 180,E1 -1038.689,E2 -1038.689} C_VEL
LIN {X 0,Y 728.151,Z 194.534,A -85,B 0,C 180,E1 -1041.637,E2 -1041.637} C_VEL
LIN {X 0,Y 728.155,Z 194.521,A -85,B 0,C 180,E1 -1044.682,E2 -1044.682} C_VEL
LIN {X 0,Y 728.156,Z 194.53,A -85,B 0,C 180,E1 -1047.712,E2 -1047.712} C_VEL
LIN {X 0,Y 728.158,Z 194.519,A -85,B 0,C 180,E1 -1050.735,E2 -1050.735} C_VEL
LIN {X 0,Y 728.155,Z 194.534,A -85,B 0,C 180,E1 -1053.758,E2 -1053.758} C_VEL
LIN {X 0,Y 728.157,Z 194.516,A -85,B 0,C 180,E1 -1056.79,E2 -1056.79} C_VEL
LIN {X 0,Y 728.155,Z 194.53,A -85,B 0,C 180,E1 -1059.838,E2 -1059.838} C_VEL
LIN {X 0,Y 728.156,Z 194.517,A -85,B 0,C 180,E1 -1062.888,E2 -1062.888} C_VEL
LIN {X 0,Y 728.156,Z 194.529,A -85,B 0,C 180,E1 -1065.852,E2 -1065.852} C_VEL
LIN {X 0,Y 728.157,Z 194.518,A -85,B 0,C 180,E1 -1068.916,E2 -1068.916} C_VEL
LIN {X 0,Y 728.148,Z 194.529,A -85,B 0,C 180,E1 -1071.948,E2 -1071.948} C_VEL
LIN {X 0,Y 728.155,Z 194.517,A -85,B 0,C 180,E1 -1074.958,E2 -1074.958} C_VEL
LIN {X 0,Y 728.148,Z 194.531,A -85,B 0,C 180,E1 -1077.954,E2 -1077.954} C_VEL
LIN {X 0,Y 728.155,Z 194.515,A -85,B 0,C 180,E1 -1080.944,E2 -1080.944} C_VEL
LIN {X 0,Y 728.143,Z 194.531,A -85,B 0,C 180,E1 -1084.016,E2 -1084.016} C_VEL
LIN {X 0,Y 728.147,Z 194.516,A -85,B 0,C 180,E1 -1086.941,E2 -1086.941} C_VEL
LIN {X 0,Y 728.141,Z 194.531,A -85,B 0,C 180,E1 -1090.044,E2 -1090.044} C_VEL
LIN {X 0,Y 728.139,Z 194.522,A -85,B 0,C 180,E1 -1092.934,E2 -1092.934} C_VEL
LIN {X 0,Y 728.142,Z 194.532,A -85,B 0,C 180,E1 -1096.023,E2 -1096.023} C_VEL
LIN {X 0,Y 728.128,Z 194.523,A -85,B 0,C 180,E1 -1098.887,E2 -1098.887} C_VEL
LIN {X 0,Y 728.155,Z 194.533,A -85,B 0,C 180,E1 -1101.932,E2 -1101.932} C_VEL
LIN {X 0,Y 728.114,Z 194.526,A -85,B 0,C 180,E1 -1104.762,E2 -1104.762} C_VEL
LIN {X 0,Y 728.154,Z 194.527,A -85,B 0,C 180,E1 -1107.662,E2 -1107.662} C_VEL
LIN {X 0,Y 728.111,Z 194.53,A -85,B 0,C 180,E1 -1110.447,E2 -1110.447} C_VEL
LIN {X 0,Y 728.146,Z 194.524,A -85,B 0,C 180,E1 -1113.251,E2 -1113.251} C_VEL
LIN {X 0,Y 728.12,Z 194.531,A -85,B 0,C 180,E1 -1116.29,E2 -1116.29} C_VEL
LIN {X 0,Y 728.111,Z 194.527,A -85,B 0,C 180,E1 -1118.989,E2 -1118.989} C_VEL
LIN {X 0,Y 728.154,Z 194.532,A -85,B 0,C 180,E1 -1121.97,E2 -1121.97} C_VEL
LIN {X 0,Y 728.098,Z 194.53,A -85,B 0,C 180,E1 -1124.679,E2 -1124.679} C_VEL
LIN {X 0,Y 728.142,Z 194.528,A -85,B 0,C 180,E1 -1127.395,E2 -1127.395} C_VEL
LIN {X 0,Y 728.107,Z 194.53,A -85,B 0,C 180,E1 -1130.417,E2 -1130.417} C_VEL
LIN {X 0,Y 728.128,Z 194.767,A -85,B 0,C 180,E1 -1130.668,E2 -1130.668} C_VEL
LIN {X 0,Y 729.397,Z 198.009,A -85,B 0,C 180,E1 -1130.906,E2 -1130.906} C_VEL
LIN {X 0,Y 733.184,Z 205.799,A -85,B 0,C 180,E1 -1131.518,E2 -1131.518} C_VEL
LIN {X 0,Y 732.67,Z 253.703,A -85,B 0,C 180,E1 -1133.734,E2 -1133.734} C_VEL
LIN {X 0,Y 732.316,Z 299.265,A -85,B 0,C 180,E1 -1135.771,E2 -1135.771} C_VEL
LIN {X 0,Y 733.106,Z 305.86,A -85,B 0,C 180,E1 -1135.89,E2 -1135.89} C_VEL
LIN {X 0,Y 732.282,Z 568.349,A -85,B 0,C 180,E1 -1138.842,E2 -1138.842} C_VEL
LIN {X 0,Y 731.89,Z 690.853,A -85,B 0,C 180,E1 -1140.213,E2 -1140.213} C_VEL
LIN {X 0,Y 731.647,Z 716.249,A -85,B 0,C 180,E1 -1140.638,E2 -1140.638} C_VEL
LIN {X 0,Y 731.424,Z 737.796,A -85,B 0,C 180,E1 -1141.133,E2 -1141.133} C_VEL
LIN {X 0,Y 731.146,Z 761.29,A -85,B 0,C 180,E1 -1141.804,E2 -1141.804} C_VEL
LIN {X 0,Y 730.784,Z 784.275,A -85,B 0,C 180,E1 -1142.622,E2 -1142.622} C_VEL
LIN {X 0,Y 730.482,Z 806.069,A -85,B 0,C 180,E1 -1143.535,E2 -1143.535} C_VEL
LIN {X 0,Y 730.059,Z 827.946,A -85,B 0,C 180,E1 -1144.616,E2 -1144.616} C_VEL
LIN {X 0,Y 729.744,Z 849.07,A -85,B 0,C 180,E1 -1145.815,E2 -1145.815} C_VEL
LIN {X 0,Y 729.359,Z 868.79,A -85,B 0,C 180,E1 -1147.111,E2 -1147.111} C_VEL
LIN {X 0,Y 729.072,Z 887.765,A -85,B 0,C 180,E1 -1148.52,E2 -1148.52} C_VEL
LIN {X 0,Y 728.776,Z 904.462,A -85,B 0,C 180,E1 -1149.94,E2 -1149.94} C_VEL
LIN {X 0,Y 728.573,Z 920.962,A -85,B 0,C 180,E1 -1151.517,E2 -1151.517} C_VEL
LIN {X 0,Y 728.355,Z 935.453,A -85,B 0,C 180,E1 -1153.107,E2 -1153.107} C_VEL
LIN {X 0,Y 728.207,Z 949.058,A -85,B 0,C 180,E1 -1154.796,E2 -1154.796} C_VEL
LIN {X 0,Y 728.086,Z 960.794,A -85,B 0,C 180,E1 -1156.499,E2 -1156.499} C_VEL
LIN {X 0,Y 728.025,Z 970.951,A -85,B 0,C 180,E1 -1158.192,E2 -1158.192} C_VEL
LIN {X 0,Y 727.958,Z 980.182,A -85,B 0,C 180,E1 -1160.034,E2 -1160.034} C_VEL
LIN {X 0,Y 727.923,Z 986.815,A -85,B 0,C 180,E1 -1161.628,E2 -1161.628} C_VEL
LIN {X 0,Y 727.91,Z 993.245,A -85,B 0,C 180,E1 -1163.533,E2 -1163.533} C_VEL
LIN {X 0,Y 727.917,Z 997.813,A -85,B 0,C 180,E1 -1165.43,E2 -1165.43} C_VEL
LIN {X 0,Y 727.882,Z 1000.684,A -85,B 0,C 180,E1 -1167.165,E2 -1167.165} C_VEL
LIN {X 0,Y 727.89,Z 1002.262,A -85,B 0,C 180,E1 -1169.134,E2 -1169.134} C_VEL
LIN {X 0,Y 727.883,Z 1002.306,A -85,B 0,C 180,E1 -1170.708,E2 -1170.708} C_VEL
LIN {X 0,Y 727.89,Z 1001.017,A -85,B 0,C 180,E1 -1172.598,E2 -1172.598} C_VEL
LIN {X 0,Y 727.915,Z 997.971,A -85,B 0,C 180,E1 -1174.491,E2 -1174.491} C_VEL
LIN {X 0,Y 727.915,Z 993.864,A -85,B 0,C 180,E1 -1176.23,E2 -1176.23} C_VEL
LIN {X 0,Y 727.937,Z 987.422,A -85,B 0,C 180,E1 -1178.213,E2 -1178.213} C_VEL
LIN {X 0,Y 727.95,Z 980.891,A -85,B 0,C 180,E1 -1179.807,E2 -1179.807} C_VEL
LIN {X 0,Y 728.027,Z 971.868,A -85,B 0,C 180,E1 -1181.648,E2 -1181.648} C_VEL
LIN {X 0,Y 728.079,Z 961.315,A -85,B 0,C 180,E1 -1183.42,E2 -1183.42} C_VEL
LIN {X 0,Y 728.191,Z 950.217,A -85,B 0,C 180,E1 -1185.042,E2 -1185.042} C_VEL
LIN {X 0,Y 728.355,Z 936.633,A -85,B 0,C 180,E1 -1186.756,E2 -1186.756} C_VEL
LIN {X 0,Y 728.512,Z 923.292,A -85,B 0,C 180,E1 -1188.236,E2 -1188.236} C_VEL
LIN {X 0,Y 728.757,Z 906.319,A -85,B 0,C 180,E1 -1189.893,E2 -1189.893} C_VEL
LIN {X 0,Y 729.028,Z 889.791,A -85,B 0,C 180,E1 -1191.313,E2 -1191.313} C_VEL
LIN {X 0,Y 729.342,Z 870.252,A -85,B 0,C 180,E1 -1192.786,E2 -1192.786} C_VEL
LIN {X 0,Y 729.683,Z 851.761,A -85,B 0,C 180,E1 -1194.015,E2 -1194.015} C_VEL
LIN {X 0,Y 730.033,Z 830.348,A -85,B 0,C 180,E1 -1195.255,E2 -1195.255} C_VEL
LIN {X 0,Y 730.388,Z 810.156,A -85,B 0,C 180,E1 -1196.274,E2 -1196.274} C_VEL
LIN {X 0,Y 730.764,Z 786.714,A -85,B 0,C 180,E1 -1197.282,E2 -1197.282} C_VEL
LIN {X 0,Y 731.014,Z 766.425,A -85,B 0,C 180,E1 -1198.024,E2 -1198.024} C_VEL
LIN {X 0,Y 731.408,Z 740.95,A -85,B 0,C 180,E1 -1198.786,E2 -1198.786} C_VEL
LIN {X 0,Y 731.62,Z 719.758,A -85,B 0,C 180,E1 -1199.287,E2 -1199.287} C_VEL
LIN {X 0,Y 731.875,Z 695.743,A -85,B 0,C 180,E1 -1199.723,E2 -1199.723} C_VEL
LIN {X 0,Y 732.027,Z 654.274,A -85,B 0,C 180,E1 -1200.21,E2 -1200.21} C_VEL
LIN {X 0,Y 732.741,Z 411.97,A -85,B 0,C 180,E1 -1202.908,E2 -1202.908} C_VEL
LIN {X 0,Y 732.91,Z 302.894,A -85,B 0,C 180,E1 -1204.155,E2 -1204.155} C_VEL
LIN {X 0,Y 732.215,Z 298.171,A -85,B 0,C 180,E1 -1204.261,E2 -1204.261} C_VEL
LIN {X 0,Y 732.862,Z 239.016,A -85,B 0,C 180,E1 -1206.937,E2 -1206.937} C_VEL
LIN {X 0,Y 733.177,Z 205.822,A -85,B 0,C 180,E1 -1208.481,E2 -1208.481} C_VEL
LIN {X 0,Y 729.325,Z 197.843,A -85,B 0,C 180,E1 -1209.106,E2 -1209.106} C_VEL
LIN {X 0,Y 728.113,Z 194.537,A -85,B 0,C 180,E1 -1209.362,E2 -1209.362} C_VEL
LIN {X 0,Y 728.154,Z 194.53,A -85,B 0,C 180,E1 -1212.256,E2 -1212.256} C_VEL
LIN {X 0,Y 728.109,Z 194.535,A -85,B 0,C 180,E1 -1215.233,E2 -1215.233} C_VEL
LIN {X 0,Y 728.139,Z 194.532,A -85,B 0,C 180,E1 -1217.98,E2 -1217.98} C_VEL
LIN {X 0,Y 728.123,Z 194.534,A -85,B 0,C 180,E1 -1220.926,E2 -1220.926} C_VEL
LIN {X 0,Y 728.13,Z 194.534,A -85,B 0,C 180,E1 -1223.715,E2 -1223.715} C_VEL
LIN {X 0,Y 728.19,Z 194.734,A -85,B 0,C 180,E1 -1226.522,E2 -1226.522} C_VEL
LIN {X 0,Y 731.371,Z 203.57,A -85,B 0,C 180,E1 -1227.224,E2 -1227.224} C_VEL
LIN {X 0,Y 730.574,Z 253.886,A -85,B 0,C 180,E1 -1230.07,E2 -1230.07} C_VEL
LIN {X 0,Y 730.055,Z 312.143,A -85,B 0,C 180,E1 -1233.251,E2 -1233.251} C_VEL
LIN {X 0,Y 729.76,Z 365.856,A -85,B 0,C 180,E1 -1236.116,E2 -1236.116} C_VEL
LIN {X 0,Y 729.374,Z 419.681,A -85,B 0,C 180,E1 -1238.95,E2 -1238.95} C_VEL
LIN {X 0,Y 729.027,Z 470.287,A -85,B 0,C 180,E1 -1241.576,E2 -1241.576} C_VEL
LIN {X 0,Y 729.415,Z 478.267,A -85,B 0,C 180,E1 -1241.667,E2 -1241.667} C_VEL
LIN {X 0,Y 729.12,Z 679.864,A -85,B 0,C 180,E1 -1243.719,E2 -1243.719} C_VEL
LIN {X 0,Y 729.021,Z 698.948,A -85,B 0,C 180,E1 -1244.063,E2 -1244.063} C_VEL
LIN {X 0,Y 728.904,Z 717.095,A -85,B 0,C 180,E1 -1244.536,E2 -1244.536} C_VEL
LIN {X 0,Y 728.748,Z 734.427,A -85,B 0,C 180,E1 -1245.133,E2 -1245.133} C_VEL
LIN {X 0,Y 728.624,Z 751.176,A -85,B 0,C 180,E1 -1245.861,E2 -1245.861} C_VEL
LIN {X 0,Y 728.479,Z 766.812,A -85,B 0,C 180,E1 -1246.694,E2 -1246.694} C_VEL
LIN {X 0,Y 728.334,Z 781.987,A -85,B 0,C 180,E1 -1247.674,E2 -1247.674} C_VEL
LIN {X 0,Y 728.205,Z 795.921,A -85,B 0,C 180,E1 -1248.756,E2 -1248.756} C_VEL
LIN {X 0,Y 728.1,Z 808.747,A -85,B 0,C 180,E1 -1249.956,E2 -1249.956} C_VEL
LIN {X 0,Y 728.023,Z 820.005,A -85,B 0,C 180,E1 -1251.231,E2 -1251.231} C_VEL
LIN {X 0,Y 727.969,Z 829.898,A -85,B 0,C 180,E1 -1252.61,E2 -1252.61} C_VEL
LIN {X 0,Y 727.939,Z 837.852,A -85,B 0,C 180,E1 -1254.008,E2 -1254.008} C_VEL
LIN {X 0,Y 727.919,Z 844.042,A -85,B 0,C 180,E1 -1255.43,E2 -1255.43} C_VEL
LIN {X 0,Y 727.915,Z 848.464,A -85,B 0,C 180,E1 -1256.85,E2 -1256.85} C_VEL
LIN {X 0,Y 727.911,Z 851.339,A -85,B 0,C 180,E1 -1258.347,E2 -1258.347} C_VEL
LIN {X 0,Y 727.912,Z 852.449,A -85,B 0,C 180,E1 -1259.843,E2 -1259.843} C_VEL
LIN {X 0,Y 727.913,Z 851.82,A -85,B 0,C 180,E1 -1261.338,E2 -1261.338} C_VEL
LIN {X 0,Y 727.913,Z 849.437,A -85,B 0,C 180,E1 -1262.835,E2 -1262.835} C_VEL
LIN {X 0,Y 727.921,Z 845.235,A -85,B 0,C 180,E1 -1264.333,E2 -1264.333} C_VEL
LIN {X 0,Y 727.931,Z 839.464,A -85,B 0,C 180,E1 -1265.755,E2 -1265.755} C_VEL
LIN {X 0,Y 727.968,Z 831.804,A -85,B 0,C 180,E1 -1267.18,E2 -1267.18} C_VEL
LIN {X 0,Y 728.012,Z 822.466,A -85,B 0,C 180,E1 -1268.549,E2 -1268.549} C_VEL
